KUKA KRL program: EPS_2_25694_RR03_A_20260114065913.src

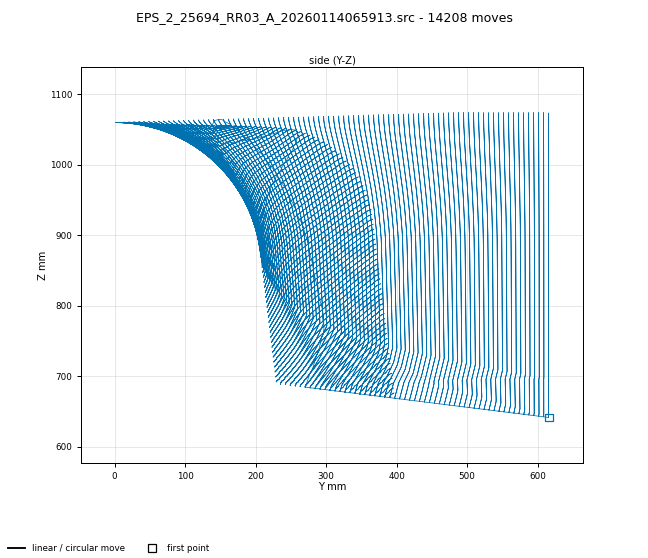
[picture p0: tool path of EPS_2_25694_RR03_A_20260114065913.src, 14208 of 14210 moves have a stored position in this frame; points joined in program order, loops and branches not executed]
&ACCESS RVP
&REL 4
&COMMENT QRS 19112012
&PARAM EDITMASK = *
DEF PART()
EXT BAS (BAS_COMMAND :IN,REAL :IN )
INT I
BAS (#INITMOV,0 )

;KUKA QRS Post kuka4.cps  Date:22-06-2017 !

File_ID=2964

QRS_PRE_INIT()

;Init var - Until changes are made in qrs_pre_init
Outlet_Square_prg=0
Inlet_1_Square_prg=0
Inlet_2_Square_prg=0
Inlet_3_Square_prg=0
Inlet_4_Square_prg=0
Inlet_5_Square_prg=0

Outlet_1={X 0.000, Y 484.060, Z 891.000, B 0.000, E1 0.000 }
Inlet_1={X 0.000, Y 496.780, Z 866.000, B 0.000, E1 180.000 }
Outlet_1_type=366
Inlet_1_type=0
;QRS#1=Sidecore dimensions
;QRS#2=375-15" PVC SDR 35
;QRS#3=DeadEnd 366
;QRS#4=
;QRS#5=
;QRS#6=
;QRS#7=
;QRS#8=
;QRS#9=20Y PSX
;QRS#10=

;QRS#11=
;QRS#12=
;QRS#13=
;QRS#14=
;QRS#15=
;QRS#16=1220x127x1372 4,5'
;QRS#17=EPS Height
;QRS#18=1074
;QRS#19=*
;QRS#20= UPDATED VERSION 22-06-2017
;QRS#21=*
Outlet_Square=0250
Inlet_1_Square=00
Inlet_2_Square=0
Inlet_3_Square=0
Inlet_4_Square=0
Inlet_5_Square=0
Mill_Square=1
Outlet_Square_Prg=252
Inlet_1_Square_prg=0

QRS_INIT()

$ADVANCE=5

; T1
PTP {E1 173.414,E2 173.414}
PTP {X 0,Y 615.481,A -85,B 0,C 180,E1 173.414,E2 173.414,E3 0,E4 0,E5 0,E6 0}
QRS_SPEED_INIT()
LIN {X 0,Y 615.481,Z 641.494,A -85,B 0,C 180,E1 173.414,E2 173.414,E3 0,E4 0,E5 0,E6 0} C_VEL
LIN {X 0,Y 615.482,Z 641.499,A -85,B 0,C 180,E1 170.801,E2 170.801} C_VEL
LIN {X 0,Y 615.492,Z 641.513,A -85,B 0,C 180,E1 168.14,E2 168.14} C_VEL
LIN {X 0,Y 615.474,Z 641.499,A -85,B 0,C 180,E1 165.451,E2 165.451} C_VEL
LIN {X 0,Y 615.49,Z 641.493,A -85,B 0,C 180,E1 162.73,E2 162.73} C_VEL
LIN {X 0,Y 615.49,Z 641.509,A -85,B 0,C 180,E1 159.968,E2 159.968} C_VEL
LIN {X 0,Y 615.475,Z 641.5,A -85,B 0,C 180,E1 157.155,E2 157.155} C_VEL
LIN {X 0,Y 615.494,Z 641.492,A -85,B 0,C 180,E1 154.427,E2 154.427} C_VEL
LIN {X 0,Y 615.492,Z 641.512,A -85,B 0,C 180,E1 151.546,E2 151.546} C_VEL
LIN {X 0,Y 615.475,Z 641.502,A -85,B 0,C 180,E1 148.913,E2 148.913} C_VEL
LIN {X 0,Y 615.48,Z 641.495,A -85,B 0,C 180,E1 146.465,E2 146.465} C_VEL
LIN {X 0,Y 615.492,Z 641.491,A -85,B 0,C 180,E1 144.164,E2 144.164} C_VEL
LIN {X 0,Y 615.485,Z 641.494,A -85,B 0,C 180,E1 141.932,E2 141.932} C_VEL
LIN {X 0,Y 615.479,Z 641.503,A -85,B 0,C 180,E1 139.393,E2 139.393} C_VEL
LIN {X 0,Y 615.494,Z 641.508,A -85,B 0,C 180,E1 136.757,E2 136.757} C_VEL
LIN {X 0,Y 615.476,Z 641.496,A -85,B 0,C 180,E1 133.997,E2 133.997} C_VEL
LIN {X 0,Y 615.478,Z 641.502,A -85,B 0,C 180,E1 131.094,E2 131.094} C_VEL
LIN {X 0,Y 615.48,Z 641.505,A -85,B 0,C 180,E1 128.904,E2 128.904} C_VEL
LIN {X 0,Y 615.485,Z 641.514,A -85,B 0,C 180,E1 126.424,E2 126.424} C_VEL
LIN {X 0,Y 615.482,Z 641.494,A -85,B 0,C 180,E1 123.534,E2 123.534} C_VEL
LIN {X 0,Y 615.481,Z 641.496,A -85,B 0,C 180,E1 120.919,E2 120.919} C_VEL
LIN {X 0,Y 615.477,Z 641.506,A -85,B 0,C 180,E1 118.45,E2 118.45} C_VEL
LIN {X 0,Y 615.477,Z 641.505,A -85,B 0,C 180,E1 115.715,E2 115.715} C_VEL
LIN {X 0,Y 615.486,Z 641.493,A -85,B 0,C 180,E1 112.844,E2 112.844} C_VEL
LIN {X 0,Y 615.483,Z 641.507,A -85,B 0,C 180,E1 110.032,E2 110.032} C_VEL
LIN {X 0,Y 615.476,Z 641.503,A -85,B 0,C 180,E1 107.27,E2 107.27} C_VEL
LIN {X 0,Y 615.488,Z 641.492,A -85,B 0,C 180,E1 104.549,E2 104.549} C_VEL
LIN {X 0,Y 615.477,Z 641.504,A -85,B 0,C 180,E1 101.861,E2 101.861} C_VEL
LIN {X 0,Y 615.487,Z 641.508,A -85,B 0,C 180,E1 99.199,E2 99.199} C_VEL
LIN {X 0,Y 615.479,Z 641.496,A -85,B 0,C 180,E1 96.557,E2 96.557} C_VEL
LIN {X 0,Y 615.483,Z 641.495,A -85,B 0,C 180,E1 93.928,E2 93.928} C_VEL
LIN {X 0,Y 615.481,Z 641.507,A -85,B 0,C 180,E1 91.309,E2 91.309} C_VEL
LIN {X 0,Y 615.481,Z 641.507,A -85,B 0,C 180,E1 88.691,E2 88.691} C_VEL
LIN {X 0,Y 615.483,Z 641.495,A -85,B 0,C 180,E1 86.072,E2 86.072} C_VEL
LIN {X 0,Y 615.478,Z 641.497,A -85,B 0,C 180,E1 83.425,E2 83.425} C_VEL
LIN {X 0,Y 615.487,Z 641.508,A -85,B 0,C 180,E1 80.801,E2 80.801} C_VEL
LIN {X 0,Y 615.477,Z 641.504,A -85,B 0,C 180,E1 78.139,E2 78.139} C_VEL
LIN {X 0,Y 615.488,Z 641.492,A -85,B 0,C 180,E1 75.451,E2 75.451} C_VEL
LIN {X 0,Y 615.476,Z 641.503,A -85,B 0,C 180,E1 72.73,E2 72.73} C_VEL
LIN {X 0,Y 615.483,Z 641.507,A -85,B 0,C 180,E1 69.968,E2 69.968} C_VEL
LIN {X 0,Y 615.486,Z 641.493,A -85,B 0,C 180,E1 67.156,E2 67.156} C_VEL
LIN {X 0,Y 615.477,Z 641.505,A -85,B 0,C 180,E1 64.285,E2 64.285} C_VEL
LIN {X 0,Y 615.48,Z 641.505,A -85,B 0,C 180,E1 61.55,E2 61.55} C_VEL
LIN {X 0,Y 615.49,Z 641.492,A -85,B 0,C 180,E1 58.913,E2 58.913} C_VEL
LIN {X 0,Y 615.482,Z 641.494,A -85,B 0,C 180,E1 56.466,E2 56.466} C_VEL
LIN {X 0,Y 615.485,Z 641.514,A -85,B 0,C 180,E1 53.576,E2 53.576} C_VEL
LIN {X 0,Y 615.478,Z 641.501,A -85,B 0,C 180,E1 50.938,E2 50.938} C_VEL
LIN {X 0,Y 615.487,Z 641.494,A -85,B 0,C 180,E1 48.527,E2 48.527} C_VEL
LIN {X 0,Y 615.473,Z 641.499,A -85,B 0,C 180,E1 45.851,E2 45.851} C_VEL
LIN {X 0,Y 615.489,Z 641.513,A -85,B 0,C 180,E1 43.049,E2 43.049} C_VEL
LIN {X 0,Y 615.497,Z 641.49,A -85,B 0,C 180,E1 40.092,E2 40.092} C_VEL
LIN {X 0,Y 615.479,Z 641.503,A -85,B 0,C 180,E1 37.242,E2 37.242} C_VEL
LIN {X 0,Y 615.491,Z 641.512,A -85,B 0,C 180,E1 34.703,E2 34.703} C_VEL
LIN {X 0,Y 615.487,Z 641.493,A -85,B 0,C 180,E1 31.685,E2 31.685} C_VEL
LIN {X 0,Y 615.482,Z 641.494,A -85,B 0,C 180,E1 29.406,E2 29.406} C_VEL
LIN {X 0,Y 615.494,Z 641.513,A -85,B 0,C 180,E1 26.443,E2 26.443} C_VEL
LIN {X 0,Y 615.488,Z 641.494,A -85,B 0,C 180,E1 23.556,E2 23.556} C_VEL
LIN {X 0,Y 615.475,Z 641.5,A -85,B 0,C 180,E1 20.731,E2 20.731} C_VEL
LIN {X 0,Y 615.488,Z 641.51,A -85,B 0,C 180,E1 17.957,E2 17.957} C_VEL
LIN {X 0,Y 615.489,Z 641.493,A -85,B 0,C 180,E1 15.226,E2 15.226} C_VEL
LIN {X 0,Y 615.475,Z 641.498,A -85,B 0,C 180,E1 12.53,E2 12.53} C_VEL
LIN {X 0,Y 615.495,Z 641.509,A -85,B 0,C 180,E1 9.862,E2 9.862} C_VEL
LIN {X 0,Y 615.481,Z 641.501,A -85,B 0,C 180,E1 7.216,E2 7.216} C_VEL
LIN {X 0,Y 615.492,Z 641.492,A -85,B 0,C 180,E1 4.584,E2 4.584} C_VEL
LIN {X 0,Y 615.476,Z 641.5,A -85,B 0,C 180,E1 1.963,E2 1.963} C_VEL
LIN {X 0,Y 615.492,Z 641.514,A -85,B 0,C 180,E1 -0.654,E2 -0.654} C_VEL
LIN {X 0,Y 615.482,Z 641.5,A -85,B 0,C 180,E1 -3.273,E2 -3.273} C_VEL
LIN {X 0,Y 615.486,Z 641.493,A -85,B 0,C 180,E1 -5.899,E2 -5.899} C_VEL
LIN {X 0,Y 615.479,Z 641.501,A -85,B 0,C 180,E1 -8.537,E2 -8.537} C_VEL
LIN {X 0,Y 615.488,Z 641.511,A -85,B 0,C 180,E1 -11.193,E2 -11.193} C_VEL
LIN {X 0,Y 615.493,Z 641.493,A -85,B 0,C 180,E1 -13.941,E2 -13.941} C_VEL
LIN {X 0,Y 615.475,Z 641.497,A -85,B 0,C 180,E1 -16.587,E2 -16.587} C_VEL
LIN {X 0,Y 615.492,Z 641.51,A -85,B 0,C 180,E1 -19.338,E2 -19.338} C_VEL
LIN {X 0,Y 615.491,Z 641.493,A -85,B 0,C 180,E1 -22.35,E2 -22.35} C_VEL
LIN {X 0,Y 615.475,Z 641.498,A -85,B 0,C 180,E1 -24.992,E2 -24.992} C_VEL
LIN {X 0,Y 615.475,Z 641.5,A -85,B 0,C 180,E1 -27.178,E2 -27.178} C_VEL
LIN {X 0,Y 615.495,Z 641.512,A -85,B 0,C 180,E1 -29.798,E2 -29.798} C_VEL
LIN {X 0,Y 615.484,Z 641.499,A -85,B 0,C 180,E1 -32.458,E2 -32.458} C_VEL
LIN {X 0,Y 615.495,Z 641.492,A -85,B 0,C 180,E1 -34.814,E2 -34.814} C_VEL
LIN {X 0,Y 615.479,Z 641.495,A -85,B 0,C 180,E1 -37.243,E2 -37.243} C_VEL
LIN {X 0,Y 615.498,Z 641.506,A -85,B 0,C 180,E1 -40.092,E2 -40.092} C_VEL
LIN {X 0,Y 615.486,Z 641.495,A -85,B 0,C 180,E1 -43.049,E2 -43.049} C_VEL
LIN {X 0,Y 615.473,Z 641.499,A -85,B 0,C 180,E1 -45.851,E2 -45.851} C_VEL
LIN {X 0,Y 615.49,Z 641.511,A -85,B 0,C 180,E1 -48.528,E2 -48.528} C_VEL
LIN {X 0,Y 615.482,Z 641.502,A -85,B 0,C 180,E1 -51.096,E2 -51.096} C_VEL
LIN {X 0,Y 615.485,Z 641.494,A -85,B 0,C 180,E1 -53.576,E2 -53.576} C_VEL
LIN {X 0,Y 615.482,Z 641.5,A -85,B 0,C 180,E1 -56.466,E2 -56.466} C_VEL
LIN {X 0,Y 615.492,Z 641.512,A -85,B 0,C 180,E1 -59.081,E2 -59.081} C_VEL
LIN {X 0,Y 615.499,Z 641.611,A -85,B 0,C 180,E1 -61.157,E2 -61.157} C_VEL
LIN {X 0,Y 615.495,Z 642.282,A -85,B 0,C 180,E1 -61.343,E2 -61.343} C_VEL
LIN {X 0,Y 615.494,Z 664.074,A -85,B 0,C 180,E1 -64.104,E2 -64.104} C_VEL
LIN {X 0,Y 615.485,Z 687.394,A -85,B 0,C 180,E1 -66.978,E2 -66.978} C_VEL
LIN {X 0,Y 615.494,Z 696.002,A -85,B 0,C 180,E1 -67.997,E2 -67.997} C_VEL
LIN {X 0,Y 615.487,Z 889.623,A -85,B 0,C 180,E1 -70.381,E2 -70.381} C_VEL
LIN {X 0,Y 615.478,Z 906.235,A -85,B 0,C 180,E1 -70.641,E2 -70.641} C_VEL
LIN {X 0,Y 615.481,Z 921.941,A -85,B 0,C 180,E1 -71.009,E2 -71.009} C_VEL
LIN {X 0,Y 615.492,Z 937.98,A -85,B 0,C 180,E1 -71.515,E2 -71.515} C_VEL
LIN {X 0,Y 615.487,Z 955.003,A -85,B 0,C 180,E1 -72.215,E2 -72.215} C_VEL
LIN {X 0,Y 615.498,Z 970.011,A -85,B 0,C 180,E1 -72.987,E2 -72.987} C_VEL
LIN {X 0,Y 615.497,Z 983.749,A -85,B 0,C 180,E1 -73.83,E2 -73.83} C_VEL
LIN {X 0,Y 615.496,Z 997.894,A -85,B 0,C 180,E1 -74.859,E2 -74.859} C_VEL
LIN {X 0,Y 615.496,Z 1010.178,A -85,B 0,C 180,E1 -75.911,E2 -75.911} C_VEL
LIN {X 0,Y 615.493,Z 1022.325,A -85,B 0,C 180,E1 -77.135,E2 -77.135} C_VEL
LIN {X 0,Y 615.491,Z 1033.537,A -85,B 0,C 180,E1 -78.474,E2 -78.474} C_VEL
LIN {X 0,Y 615.493,Z 1042.917,A -85,B 0,C 180,E1 -79.806,E2 -79.806} C_VEL
LIN {X 0,Y 615.495,Z 1050.708,A -85,B 0,C 180,E1 -81.133,E2 -81.133} C_VEL
LIN {X 0,Y 615.494,Z 1057.212,A -85,B 0,C 180,E1 -82.455,E2 -82.455} C_VEL
LIN {X 0,Y 615.494,Z 1062.49,A -85,B 0,C 180,E1 -83.773,E2 -83.773} C_VEL
LIN {X 0,Y 615.497,Z 1065.74,A -85,B 0,C 180,E1 -84.759,E2 -84.759} C_VEL
LIN {X 0,Y 615.492,Z 1069.077,A -85,B 0,C 180,E1 -86.072,E2 -86.072} C_VEL
LIN {X 0,Y 615.484,Z 1071.504,A -85,B 0,C 180,E1 -87.382,E2 -87.382} C_VEL
LIN {X 0,Y 615.494,Z 1072.869,A -85,B 0,C 180,E1 -88.691,E2 -88.691} C_VEL
LIN {X 0,Y 615.489,Z 1073.39,A -85,B 0,C 180,E1 -90,E2 -90} C_VEL
LIN {X 0,Y 615.494,Z 1072.869,A -85,B 0,C 180,E1 -91.309,E2 -91.309} C_VEL
LIN {X 0,Y 615.484,Z 1071.504,A -85,B 0,C 180,E1 -92.618,E2 -92.618} C_VEL
LIN {X 0,Y 615.492,Z 1069.077,A -85,B 0,C 180,E1 -93.928,E2 -93.928} C_VEL
LIN {X 0,Y 615.496,Z 1065.74,A -85,B 0,C 180,E1 -95.241,E2 -95.241} C_VEL
LIN {X 0,Y 615.495,Z 1059.981,A -85,B 0,C 180,E1 -96.898,E2 -96.898} C_VEL
LIN {X 0,Y 615.491,Z 1052.502,A -85,B 0,C 180,E1 -98.536,E2 -98.536} C_VEL
LIN {X 0,Y 615.489,Z 1043.967,A -85,B 0,C 180,E1 -100.028,E2 -100.028} C_VEL
LIN {X 0,Y 615.496,Z 1034.768,A -85,B 0,C 180,E1 -101.359,E2 -101.359} C_VEL
LIN {X 0,Y 615.494,Z 1025.294,A -85,B 0,C 180,E1 -102.53,E2 -102.53} C_VEL
LIN {X 0,Y 615.495,Z 1014.218,A -85,B 0,C 180,E1 -103.705,E2 -103.705} C_VEL
LIN {X 0,Y 615.495,Z 1002.119,A -85,B 0,C 180,E1 -104.802,E2 -104.802} C_VEL
LIN {X 0,Y 615.497,Z 987.714,A -85,B 0,C 180,E1 -105.904,E2 -105.904} C_VEL
LIN {X 0,Y 615.497,Z 973.021,A -85,B 0,C 180,E1 -106.842,E2 -106.842} C_VEL
LIN {X 0,Y 615.497,Z 958.52,A -85,B 0,C 180,E1 -107.613,E2 -107.613} C_VEL
LIN {X 0,Y 615.486,Z 943.271,A -85,B 0,C 180,E1 -108.281,E2 -108.281} C_VEL
LIN {X 0,Y 615.488,Z 928.006,A -85,B 0,C 180,E1 -108.818,E2 -108.818} C_VEL
LIN {X 0,Y 615.476,Z 911.542,A -85,B 0,C 180,E1 -109.251,E2 -109.251} C_VEL
LIN {X 0,Y 615.484,Z 895.965,A -85,B 0,C 180,E1 -109.533,E2 -109.533} C_VEL
LIN {X 0,Y 615.492,Z 696.002,A -85,B 0,C 180,E1 -112.003,E2 -112.003} C_VEL
LIN {X 0,Y 615.475,Z 675.734,A -85,B 0,C 180,E1 -114.451,E2 -114.451} C_VEL
LIN {X 0,Y 615.495,Z 653.871,A -85,B 0,C 180,E1 -117.176,E2 -117.176} C_VEL
LIN {X 0,Y 615.496,Z 641.859,A -85,B 0,C 180,E1 -118.727,E2 -118.727} C_VEL
LIN {X 0,Y 615.478,Z 641.5,A -85,B 0,C 180,E1 -119.406,E2 -119.406} C_VEL
LIN {X 0,Y 615.473,Z 641.498,A -85,B 0,C 180,E1 -121.685,E2 -121.685} C_VEL
LIN {X 0,Y 615.479,Z 641.495,A -85,B 0,C 180,E1 -124.021,E2 -124.021} C_VEL
LIN {X 0,Y 615.486,Z 641.505,A -85,B 0,C 180,E1 -126.937,E2 -126.937} C_VEL
LIN {X 0,Y 615.484,Z 641.501,A -85,B 0,C 180,E1 -129.749,E2 -129.749} C_VEL
LIN {X 0,Y 615.479,Z 641.494,A -85,B 0,C 180,E1 -132.352,E2 -132.352} C_VEL
LIN {X 0,Y 615.485,Z 641.5,A -85,B 0,C 180,E1 -135.067,E2 -135.067} C_VEL
LIN {X 0,Y 615.495,Z 641.503,A -85,B 0,C 180,E1 -137.917,E2 -137.917} C_VEL
LIN {X 0,Y 615.479,Z 641.5,A -85,B 0,C 180,E1 -140.249,E2 -140.249} C_VEL
LIN {X 0,Y 615.487,Z 641.493,A -85,B 0,C 180,E1 -143.061,E2 -143.061} C_VEL
LIN {X 0,Y 615.494,Z 641.514,A -85,B 0,C 180,E1 -145.979,E2 -145.979} C_VEL
LIN {X 0,Y 615.488,Z 641.506,A -85,B 0,C 180,E1 -148.315,E2 -148.315} C_VEL
LIN {X 0,Y 615.482,Z 641.501,A -85,B 0,C 180,E1 -150.593,E2 -150.593} C_VEL
LIN {X 0,Y 615.474,Z 641.498,A -85,B 0,C 180,E1 -152.954,E2 -152.954} C_VEL
LIN {X 0,Y 615.489,Z 641.495,A -85,B 0,C 180,E1 -155.728,E2 -155.728} C_VEL
LIN {X 0,Y 615.492,Z 641.511,A -85,B 0,C 180,E1 -158.568,E2 -158.568} C_VEL
LIN {X 0,Y 615.476,Z 641.496,A -85,B 0,C 180,E1 -161.394,E2 -161.394} C_VEL
LIN {X 0,Y 615.487,Z 641.496,A -85,B 0,C 180,E1 -164.095,E2 -164.095} C_VEL
LIN {X 0,Y 615.495,Z 641.513,A -85,B 0,C 180,E1 -166.799,E2 -166.799} C_VEL
LIN {X 0,Y 615.474,Z 641.5,A -85,B 0,C 180,E1 -169.473,E2 -169.473} C_VEL
LIN {X 0,Y 615.486,Z 641.493,A -85,B 0,C 180,E1 -172.124,E2 -172.124} C_VEL
LIN {X 0,Y 615.482,Z 641.502,A -85,B 0,C 180,E1 -174.759,E2 -174.759} C_VEL
LIN {X 0,Y 615.495,Z 641.508,A -85,B 0,C 180,E1 -177.382,E2 -177.382} C_VEL
LIN {X 0,Y 615.475,Z 641.498,A -85,B 0,C 180,E1 -180,E2 -180} C_VEL
LIN {X 0,Y 615.492,Z 641.492,A -85,B 0,C 180,E1 -182.618,E2 -182.618} C_VEL
LIN {X 0,Y 615.482,Z 641.504,A -85,B 0,C 180,E1 -185.241,E2 -185.241} C_VEL
LIN {X 0,Y 615.481,Z 641.494,A -85,B 0,C 180,E1 -186.586,E2 -186.586} C_VEL
LIN {X 0,Y 614.804,Z 641.649,A -85,B 0,C 180,E1 -187.132,E2 -187.132} C_VEL
LIN {X 0,Y 611.968,Z 642.066,A -85,B 0,C 180,E1 -188.018,E2 -188.018} C_VEL
LIN {X 0,Y 609.577,Z 642.375,A -85,B 0,C 180,E1 -188.731,E2 -188.731} C_VEL
LIN {X 0,Y 608.545,Z 642.492,A -85,B 0,C 180,E1 -189.28,E2 -189.28} C_VEL
LIN {X 0,Y 608.458,Z 642.502,A -85,B 0,C 180,E1 -189.466,E2 -189.466} C_VEL
LIN {X 0,Y 608.462,Z 642.506,A -85,B 0,C 180,E1 -192,E2 -192} C_VEL
LIN {X 0,Y 608.466,Z 642.497,A -85,B 0,C 180,E1 -194.72,E2 -194.72} C_VEL
LIN {X 0,Y 608.455,Z 642.5,A -85,B 0,C 180,E1 -197.476,E2 -197.476} C_VEL
LIN {X 0,Y 608.461,Z 642.508,A -85,B 0,C 180,E1 -200.274,E2 -200.274} C_VEL
LIN {X 0,Y 608.482,Z 642.502,A -85,B 0,C 180,E1 -202.485,E2 -202.485} C_VEL
LIN {X 0,Y 608.449,Z 642.499,A -85,B 0,C 180,E1 -205.301,E2 -205.301} C_VEL
LIN {X 0,Y 608.441,Z 642.499,A -85,B 0,C 180,E1 -207.518,E2 -207.518} C_VEL
LIN {X 0,Y 608.465,Z 642.498,A -85,B 0,C 180,E1 -209.974,E2 -209.974} C_VEL
LIN {X 0,Y 608.458,Z 642.507,A -85,B 0,C 180,E1 -212.524,E2 -212.524} C_VEL
LIN {X 0,Y 608.443,Z 642.502,A -85,B 0,C 180,E1 -215.277,E2 -215.277} C_VEL
LIN {X 0,Y 608.465,Z 642.497,A -85,B 0,C 180,E1 -217.746,E2 -217.746} C_VEL
LIN {X 0,Y 608.471,Z 642.498,A -85,B 0,C 180,E1 -220.333,E2 -220.333} C_VEL
LIN {X 0,Y 608.48,Z 642.503,A -85,B 0,C 180,E1 -223.311,E2 -223.311} C_VEL
LIN {X 0,Y 608.461,Z 642.498,A -85,B 0,C 180,E1 -226.131,E2 -226.131} C_VEL
LIN {X 0,Y 608.45,Z 642.502,A -85,B 0,C 180,E1 -228.824,E2 -228.824} C_VEL
LIN {X 0,Y 608.461,Z 642.509,A -85,B 0,C 180,E1 -231.413,E2 -231.413} C_VEL
LIN {X 0,Y 608.469,Z 642.501,A -85,B 0,C 180,E1 -233.951,E2 -233.951} C_VEL
LIN {X 0,Y 608.459,Z 642.499,A -85,B 0,C 180,E1 -236.33,E2 -236.33} C_VEL
LIN {X 0,Y 608.473,Z 642.496,A -85,B 0,C 180,E1 -238.727,E2 -238.727} C_VEL
LIN {X 0,Y 608.464,Z 642.501,A -85,B 0,C 180,E1 -241.381,E2 -241.381} C_VEL
LIN {X 0,Y 608.437,Z 642.513,A -85,B 0,C 180,E1 -243.965,E2 -243.965} C_VEL
LIN {X 0,Y 608.466,Z 642.507,A -85,B 0,C 180,E1 -246.156,E2 -246.156} C_VEL
LIN {X 0,Y 608.455,Z 642.498,A -85,B 0,C 180,E1 -249.019,E2 -249.019} C_VEL
LIN {X 0,Y 608.447,Z 642.503,A -85,B 0,C 180,E1 -251.829,E2 -251.829} C_VEL
LIN {X 0,Y 608.463,Z 642.505,A -85,B 0,C 180,E1 -254.594,E2 -254.594} C_VEL
LIN {X 0,Y 608.473,Z 642.496,A -85,B 0,C 180,E1 -257.323,E2 -257.323} C_VEL
LIN {X 0,Y 608.449,Z 642.501,A -85,B 0,C 180,E1 -260.023,E2 -260.023} C_VEL
LIN {X 0,Y 608.461,Z 642.51,A -85,B 0,C 180,E1 -262.701,E2 -262.701} C_VEL
LIN {X 0,Y 608.446,Z 642.502,A -85,B 0,C 180,E1 -265.362,E2 -265.362} C_VEL
LIN {X 0,Y 608.46,Z 642.498,A -85,B 0,C 180,E1 -268.014,E2 -268.014} C_VEL
LIN {X 0,Y 608.47,Z 642.502,A -85,B 0,C 180,E1 -270.662,E2 -270.662} C_VEL
LIN {X 0,Y 608.48,Z 642.504,A -85,B 0,C 180,E1 -273.311,E2 -273.311} C_VEL
LIN {X 0,Y 608.452,Z 642.5,A -85,B 0,C 180,E1 -275.967,E2 -275.967} C_VEL
LIN {X 0,Y 608.454,Z 642.5,A -85,B 0,C 180,E1 -278.636,E2 -278.636} C_VEL
LIN {X 0,Y 608.472,Z 642.506,A -85,B 0,C 180,E1 -281.324,E2 -281.324} C_VEL
LIN {X 0,Y 608.464,Z 642.501,A -85,B 0,C 180,E1 -284.037,E2 -284.037} C_VEL
LIN {X 0,Y 608.475,Z 642.496,A -85,B 0,C 180,E1 -286.783,E2 -286.783} C_VEL
LIN {X 0,Y 608.443,Z 642.507,A -85,B 0,C 180,E1 -289.57,E2 -289.57} C_VEL
LIN {X 0,Y 608.47,Z 642.5,A -85,B 0,C 180,E1 -292.405,E2 -292.405} C_VEL
LIN {X 0,Y 608.452,Z 642.501,A -85,B 0,C 180,E1 -294.57,E2 -294.57} C_VEL
LIN {X 0,Y 608.482,Z 642.495,A -85,B 0,C 180,E1 -297.209,E2 -297.209} C_VEL
LIN {X 0,Y 608.464,Z 642.504,A -85,B 0,C 180,E1 -299.972,E2 -299.972} C_VEL
LIN {X 0,Y 608.46,Z 642.506,A -85,B 0,C 180,E1 -302.523,E2 -302.523} C_VEL
LIN {X 0,Y 608.438,Z 642.501,A -85,B 0,C 180,E1 -305.277,E2 -305.277} C_VEL
LIN {X 0,Y 608.46,Z 642.498,A -85,B 0,C 180,E1 -307.746,E2 -307.746} C_VEL
LIN {X 0,Y 608.447,Z 642.505,A -85,B 0,C 180,E1 -310.329,E2 -310.329} C_VEL
LIN {X 0,Y 608.466,Z 642.499,A -85,B 0,C 180,E1 -313.309,E2 -313.309} C_VEL
LIN {X 0,Y 608.468,Z 642.497,A -85,B 0,C 180,E1 -316.131,E2 -316.131} C_VEL
LIN {X 0,Y 608.456,Z 642.507,A -85,B 0,C 180,E1 -318.824,E2 -318.824} C_VEL
LIN {X 0,Y 608.471,Z 642.502,A -85,B 0,C 180,E1 -321.413,E2 -321.413} C_VEL
LIN {X 0,Y 608.471,Z 642.496,A -85,B 0,C 180,E1 -323.949,E2 -323.949} C_VEL
LIN {X 0,Y 608.458,Z 642.498,A -85,B 0,C 180,E1 -326.329,E2 -326.329} C_VEL
LIN {X 0,Y 608.466,Z 642.498,A -85,B 0,C 180,E1 -328.727,E2 -328.727} C_VEL
LIN {X 0,Y 608.474,Z 642.505,A -85,B 0,C 180,E1 -331.377,E2 -331.377} C_VEL
LIN {X 0,Y 608.471,Z 642.498,A -85,B 0,C 180,E1 -334.276,E2 -334.276} C_VEL
LIN {X 0,Y 608.444,Z 642.5,A -85,B 0,C 180,E1 -336.876,E2 -336.876} C_VEL
LIN {X 0,Y 608.459,Z 642.501,A -85,B 0,C 180,E1 -339.32,E2 -339.32} C_VEL
LIN {X 0,Y 608.448,Z 642.51,A -85,B 0,C 180,E1 -341.828,E2 -341.828} C_VEL
LIN {X 0,Y 608.472,Z 642.498,A -85,B 0,C 180,E1 -344.594,E2 -344.594} C_VEL
LIN {X 0,Y 608.466,Z 642.497,A -85,B 0,C 180,E1 -347.323,E2 -347.323} C_VEL
LIN {X 0,Y 608.46,Z 642.505,A -85,B 0,C 180,E1 -350.023,E2 -350.023} C_VEL
LIN {X 0,Y 608.475,Z 642.501,A -85,B 0,C 180,E1 -352.701,E2 -352.701} C_VEL
LIN {X 0,Y 608.46,Z 642.498,A -85,B 0,C 180,E1 -355.363,E2 -355.363} C_VEL
LIN {X 0,Y 608.447,Z 642.501,A -85,B 0,C 180,E1 -358.014,E2 -358.014} C_VEL
LIN {X 0,Y 608.484,Z 642.507,A -85,B 0,C 180,E1 -360.662,E2 -360.662} C_VEL
LIN {X 0,Y 608.474,Z 642.498,A -85,B 0,C 180,E1 -363.311,E2 -363.311} C_VEL
LIN {X 0,Y 608.481,Z 642.495,A -85,B 0,C 180,E1 -365.967,E2 -365.967} C_VEL
LIN {X 0,Y 608.45,Z 642.504,A -85,B 0,C 180,E1 -368.636,E2 -368.636} C_VEL
LIN {X 0,Y 608.474,Z 642.503,A -85,B 0,C 180,E1 -371.324,E2 -371.324} C_VEL
LIN {X 0,Y 608.458,Z 642.498,A -85,B 0,C 180,E1 -374.038,E2 -374.038} C_VEL
LIN {X 0,Y 608.467,Z 642.499,A -85,B 0,C 180,E1 -376.784,E2 -376.784} C_VEL
LIN {X 0,Y 608.454,Z 642.508,A -85,B 0,C 180,E1 -379.571,E2 -379.571} C_VEL
LIN {X 0,Y 608.468,Z 642.496,A -85,B 0,C 180,E1 -382.482,E2 -382.482} C_VEL
LIN {X 0,Y 608.448,Z 642.504,A -85,B 0,C 180,E1 -385.301,E2 -385.301} C_VEL
LIN {X 0,Y 608.444,Z 642.507,A -85,B 0,C 180,E1 -387.518,E2 -387.518} C_VEL
LIN {X 0,Y 608.471,Z 642.506,A -85,B 0,C 180,E1 -389.975,E2 -389.975} C_VEL
LIN {X 0,Y 608.457,Z 642.5,A -85,B 0,C 180,E1 -392.524,E2 -392.524} C_VEL
LIN {X 0,Y 608.443,Z 642.5,A -85,B 0,C 180,E1 -395.278,E2 -395.278} C_VEL
LIN {X 0,Y 608.469,Z 642.5,A -85,B 0,C 180,E1 -397.746,E2 -397.746} C_VEL
LIN {X 0,Y 608.474,Z 642.507,A -85,B 0,C 180,E1 -400.333,E2 -400.333} C_VEL
LIN {X 0,Y 608.48,Z 642.495,A -85,B 0,C 180,E1 -403.311,E2 -403.311} C_VEL
LIN {X 0,Y 608.462,Z 642.502,A -85,B 0,C 180,E1 -406.131,E2 -406.131} C_VEL
LIN {X 0,Y 608.454,Z 642.506,A -85,B 0,C 180,E1 -408.825,E2 -408.825} C_VEL
LIN {X 0,Y 608.463,Z 642.498,A -85,B 0,C 180,E1 -411.413,E2 -411.413} C_VEL
LIN {X 0,Y 608.471,Z 642.496,A -85,B 0,C 180,E1 -413.951,E2 -413.951} C_VEL
LIN {X 0,Y 608.459,Z 642.5,A -85,B 0,C 180,E1 -416.33,E2 -416.33} C_VEL
LIN {X 0,Y 608.476,Z 642.501,A -85,B 0,C 180,E1 -418.728,E2 -418.728} C_VEL
LIN {X 0,Y 608.508,Z 642.684,A -85,B 0,C 180,E1 -421.015,E2 -421.015} C_VEL
LIN {X 0,Y 608.742,Z 646.926,A -85,B 0,C 180,E1 -421.605,E2 -421.605} C_VEL
LIN {X 0,Y 608.689,Z 667.591,A -85,B 0,C 180,E1 -424.236,E2 -424.236} C_VEL
LIN {X 0,Y 608.628,Z 690.455,A -85,B 0,C 180,E1 -427.082,E2 -427.082} C_VEL
LIN {X 0,Y 608.66,Z 695.999,A -85,B 0,C 180,E1 -427.737,E2 -427.737} C_VEL
LIN {X 0,Y 608.923,Z 700.026,A -85,B 0,C 180,E1 -427.814,E2 -427.814} C_VEL
LIN {X 0,Y 608.793,Z 898.977,A -85,B 0,C 180,E1 -430.288,E2 -430.288} C_VEL
LIN {X 0,Y 608.766,Z 915.2,A -85,B 0,C 180,E1 -430.616,E2 -430.616} C_VEL
LIN {X 0,Y 608.751,Z 931.96,A -85,B 0,C 180,E1 -431.097,E2 -431.097} C_VEL
LIN {X 0,Y 608.685,Z 947.354,A -85,B 0,C 180,E1 -431.672,E2 -431.672} C_VEL
LIN {X 0,Y 608.673,Z 962.02,A -85,B 0,C 180,E1 -432.357,E2 -432.357} C_VEL
LIN {X 0,Y 608.616,Z 975.841,A -85,B 0,C 180,E1 -433.135,E2 -433.135} C_VEL
LIN {X 0,Y 608.578,Z 990.054,A -85,B 0,C 180,E1 -434.082,E2 -434.082} C_VEL
LIN {X 0,Y 608.556,Z 1003.132,A -85,B 0,C 180,E1 -435.111,E2 -435.111} C_VEL
LIN {X 0,Y 608.515,Z 1016.01,A -85,B 0,C 180,E1 -436.305,E2 -436.305} C_VEL
LIN {X 0,Y 608.491,Z 1026.914,A -85,B 0,C 180,E1 -437.493,E2 -437.493} C_VEL
LIN {X 0,Y 608.488,Z 1036.208,A -85,B 0,C 180,E1 -438.677,E2 -438.677} C_VEL
LIN {X 0,Y 608.464,Z 1045.26,A -85,B 0,C 180,E1 -440.023,E2 -440.023} C_VEL
LIN {X 0,Y 608.445,Z 1052.859,A -85,B 0,C 180,E1 -441.364,E2 -441.364} C_VEL
LIN {X 0,Y 608.44,Z 1060.467,A -85,B 0,C 180,E1 -443.034,E2 -443.034} C_VEL
LIN {X 0,Y 608.439,Z 1066.245,A -85,B 0,C 180,E1 -444.698,E2 -444.698} C_VEL
LIN {X 0,Y 608.429,Z 1069.633,A -85,B 0,C 180,E1 -446.026,E2 -446.026} C_VEL
LIN {X 0,Y 608.412,Z 1072.086,A -85,B 0,C 180,E1 -447.352,E2 -447.352} C_VEL
LIN {X 0,Y 608.446,Z 1073.477,A -85,B 0,C 180,E1 -448.676,E2 -448.676} C_VEL
LIN {X 0,Y 608.429,Z 1074,A -85,B 0,C 180,E1 -450,E2 -450} C_VEL
LIN {X 0,Y 608.446,Z 1073.477,A -85,B 0,C 180,E1 -451.324,E2 -451.324} C_VEL
LIN {X 0,Y 608.412,Z 1072.086,A -85,B 0,C 180,E1 -452.648,E2 -452.648} C_VEL
LIN {X 0,Y 608.429,Z 1069.633,A -85,B 0,C 180,E1 -453.974,E2 -453.974} C_VEL
LIN {X 0,Y 608.438,Z 1066.245,A -85,B 0,C 180,E1 -455.302,E2 -455.302} C_VEL
LIN {X 0,Y 608.44,Z 1060.467,A -85,B 0,C 180,E1 -456.966,E2 -456.966} C_VEL
LIN {X 0,Y 608.445,Z 1052.859,A -85,B 0,C 180,E1 -458.636,E2 -458.636} C_VEL
LIN {X 0,Y 608.458,Z 1044.248,A -85,B 0,C 180,E1 -460.145,E2 -460.145} C_VEL
LIN {X 0,Y 608.465,Z 1034.969,A -85,B 0,C 180,E1 -461.492,E2 -461.492} C_VEL
LIN {X 0,Y 608.49,Z 1025.424,A -85,B 0,C 180,E1 -462.676,E2 -462.676} C_VEL
LIN {X 0,Y 608.519,Z 1013.976,A -85,B 0,C 180,E1 -463.896,E2 -463.896} C_VEL
LIN {X 0,Y 608.553,Z 1002.147,A -85,B 0,C 180,E1 -464.975,E2 -464.975} C_VEL
LIN {X 0,Y 608.598,Z 988.893,A -85,B 0,C 180,E1 -466.004,E2 -466.004} C_VEL
LIN {X 0,Y 608.616,Z 975.841,A -85,B 0,C 180,E1 -466.865,E2 -466.865} C_VEL
LIN {X 0,Y 608.673,Z 962.02,A -85,B 0,C 180,E1 -467.643,E2 -467.643} C_VEL
LIN {X 0,Y 608.685,Z 947.354,A -85,B 0,C 180,E1 -468.328,E2 -468.328} C_VEL
LIN {X 0,Y 608.751,Z 931.96,A -85,B 0,C 180,E1 -468.903,E2 -468.903} C_VEL
LIN {X 0,Y 608.766,Z 915.2,A -85,B 0,C 180,E1 -469.384,E2 -469.384} C_VEL
LIN {X 0,Y 608.793,Z 898.977,A -85,B 0,C 180,E1 -469.712,E2 -469.712} C_VEL
LIN {X 0,Y 608.881,Z 697.149,A -85,B 0,C 180,E1 -472.224,E2 -472.224} C_VEL
LIN {X 0,Y 608.632,Z 695.447,A -85,B 0,C 180,E1 -472.309,E2 -472.309} C_VEL
LIN {X 0,Y 608.682,Z 672.819,A -85,B 0,C 180,E1 -475.107,E2 -475.107} C_VEL
LIN {X 0,Y 608.74,Z 649.498,A -85,B 0,C 180,E1 -478.064,E2 -478.064} C_VEL
LIN {X 0,Y 608.582,Z 643.159,A -85,B 0,C 180,E1 -478.896,E2 -478.896} C_VEL
LIN {X 0,Y 608.489,Z 642.596,A -85,B 0,C 180,E1 -479.018,E2 -479.018} C_VEL
LIN {X 0,Y 608.474,Z 642.501,A -85,B 0,C 180,E1 -481.315,E2 -481.315} C_VEL
LIN {X 0,Y 608.468,Z 642.498,A -85,B 0,C 180,E1 -483.734,E2 -483.734} C_VEL
LIN {X 0,Y 608.471,Z 642.496,A -85,B 0,C 180,E1 -486.089,E2 -486.089} C_VEL
LIN {X 0,Y 608.463,Z 642.498,A -85,B 0,C 180,E1 -488.587,E2 -488.587} C_VEL
LIN {X 0,Y 608.463,Z 642.509,A -85,B 0,C 180,E1 -491.342,E2 -491.342} C_VEL
LIN {X 0,Y 608.444,Z 642.5,A -85,B 0,C 180,E1 -494.263,E2 -494.263} C_VEL
LIN {X 0,Y 608.456,Z 642.5,A -85,B 0,C 180,E1 -497.041,E2 -497.041} C_VEL
LIN {X 0,Y 608.459,Z 642.509,A -85,B 0,C 180,E1 -499.697,E2 -499.697} C_VEL
LIN {X 0,Y 608.469,Z 642.5,A -85,B 0,C 180,E1 -502.254,E2 -502.254} C_VEL
LIN {X 0,Y 608.483,Z 642.495,A -85,B 0,C 180,E1 -505.088,E2 -505.088} C_VEL
LIN {X 0,Y 608.464,Z 642.506,A -85,B 0,C 180,E1 -507.905,E2 -507.905} C_VEL
LIN {X 0,Y 608.478,Z 642.505,A -85,B 0,C 180,E1 -510.221,E2 -510.221} C_VEL
LIN {X 0,Y 608.468,Z 642.499,A -85,B 0,C 180,E1 -512.792,E2 -512.792} C_VEL
LIN {X 0,Y 608.449,Z 642.499,A -85,B 0,C 180,E1 -515.429,E2 -515.429} C_VEL
LIN {X 0,Y 608.47,Z 642.505,A -85,B 0,C 180,E1 -518.308,E2 -518.308} C_VEL
LIN {X 0,Y 608.46,Z 642.499,A -85,B 0,C 180,E1 -521.283,E2 -521.283} C_VEL
LIN {X 0,Y 608.478,Z 642.496,A -85,B 0,C 180,E1 -523.907,E2 -523.907} C_VEL
LIN {X 0,Y 608.47,Z 642.505,A -85,B 0,C 180,E1 -526.644,E2 -526.644} C_VEL
LIN {X 0,Y 608.458,Z 642.502,A -85,B 0,C 180,E1 -529.35,E2 -529.35} C_VEL
LIN {X 0,Y 608.475,Z 642.495,A -85,B 0,C 180,E1 -532.033,E2 -532.033} C_VEL
LIN {X 0,Y 608.461,Z 642.501,A -85,B 0,C 180,E1 -534.698,E2 -534.698} C_VEL
LIN {X 0,Y 608.483,Z 642.505,A -85,B 0,C 180,E1 -537.352,E2 -537.352} C_VEL
LIN {X 0,Y 608.465,Z 642.498,A -85,B 0,C 180,E1 -540,E2 -540} C_VEL
LIN {X 0,Y 608.481,Z 642.495,A -85,B 0,C 180,E1 -542.648,E2 -542.648} C_VEL
LIN {X 0,Y 608.461,Z 642.504,A -85,B 0,C 180,E1 -545.302,E2 -545.302} C_VEL
LIN {X 0,Y 608.475,Z 642.502,A -85,B 0,C 180,E1 -547.967,E2 -547.967} C_VEL
LIN {X 0,Y 608.458,Z 642.502,A -85,B 0,C 180,E1 -549.466,E2 -549.466} C_VEL
LIN {X 0,Y 607.783,Z 642.59,A -85,B 0,C 180,E1 -550.019,E2 -550.019} C_VEL
LIN {X 0,Y 604.929,Z 642.946,A -85,B 0,C 180,E1 -550.916,E2 -550.916} C_VEL
LIN {X 0,Y 602.523,Z 643.245,A -85,B 0,C 180,E1 -551.637,E2 -551.637} C_VEL
LIN {X 0,Y 601.489,Z 643.371,A -85,B 0,C 180,E1 -552.194,E2 -552.194} C_VEL
LIN {X 0,Y 601.405,Z 643.378,A -85,B 0,C 180,E1 -552.383,E2 -552.383} C_VEL
LIN {X 0,Y 601.423,Z 643.374,A -85,B 0,C 180,E1 -554.897,E2 -554.897} C_VEL
LIN {X 0,Y 601.425,Z 643.374,A -85,B 0,C 180,E1 -556.986,E2 -556.986} C_VEL
LIN {X 0,Y 601.406,Z 643.381,A -85,B 0,C 180,E1 -559.809,E2 -559.809} C_VEL
LIN {X 0,Y 601.444,Z 643.376,A -85,B 0,C 180,E1 -562.681,E2 -562.681} C_VEL
LIN {X 0,Y 601.398,Z 643.38,A -85,B 0,C 180,E1 -564.878,E2 -564.878} C_VEL
LIN {X 0,Y 601.416,Z 643.376,A -85,B 0,C 180,E1 -567.867,E2 -567.867} C_VEL
LIN {X 0,Y 601.437,Z 643.375,A -85,B 0,C 180,E1 -570.163,E2 -570.163} C_VEL
LIN {X 0,Y 601.417,Z 643.386,A -85,B 0,C 180,E1 -572.717,E2 -572.717} C_VEL
LIN {X 0,Y 601.412,Z 643.379,A -85,B 0,C 180,E1 -575.116,E2 -575.116} C_VEL
LIN {X 0,Y 601.427,Z 643.376,A -85,B 0,C 180,E1 -577.419,E2 -577.419} C_VEL
LIN {X 0,Y 601.41,Z 643.376,A -85,B 0,C 180,E1 -579.995,E2 -579.995} C_VEL
LIN {X 0,Y 601.429,Z 643.378,A -85,B 0,C 180,E1 -582.668,E2 -582.668} C_VEL
LIN {X 0,Y 601.416,Z 643.382,A -85,B 0,C 180,E1 -585.483,E2 -585.483} C_VEL
LIN {X 0,Y 601.418,Z 643.375,A -85,B 0,C 180,E1 -588.407,E2 -588.407} C_VEL
LIN {X 0,Y 601.427,Z 643.376,A -85,B 0,C 180,E1 -590.876,E2 -590.876} C_VEL
LIN {X 0,Y 601.436,Z 643.381,A -85,B 0,C 180,E1 -593.734,E2 -593.734} C_VEL
LIN {X 0,Y 601.423,Z 643.374,A -85,B 0,C 180,E1 -596.687,E2 -596.687} C_VEL
LIN {X 0,Y 601.428,Z 643.375,A -85,B 0,C 180,E1 -599.059,E2 -599.059} C_VEL
LIN {X 0,Y 601.424,Z 643.378,A -85,B 0,C 180,E1 -601.374,E2 -601.374} C_VEL
LIN {X 0,Y 601.399,Z 643.384,A -85,B 0,C 180,E1 -603.637,E2 -603.637} C_VEL
LIN {X 0,Y 601.417,Z 643.378,A -85,B 0,C 180,E1 -606.59,E2 -606.59} C_VEL
LIN {X 0,Y 601.429,Z 643.375,A -85,B 0,C 180,E1 -609.479,E2 -609.479} C_VEL
LIN {X 0,Y 601.392,Z 643.39,A -85,B 0,C 180,E1 -612.312,E2 -612.312} C_VEL
LIN {X 0,Y 601.409,Z 643.388,A -85,B 0,C 180,E1 -614.409,E2 -614.409} C_VEL
LIN {X 0,Y 601.416,Z 643.376,A -85,B 0,C 180,E1 -617.172,E2 -617.172} C_VEL
LIN {X 0,Y 601.427,Z 643.375,A -85,B 0,C 180,E1 -619.905,E2 -619.905} C_VEL
LIN {X 0,Y 601.437,Z 643.383,A -85,B 0,C 180,E1 -622.615,E2 -622.615} C_VEL
LIN {X 0,Y 601.416,Z 643.379,A -85,B 0,C 180,E1 -625.308,E2 -625.308} C_VEL
LIN {X 0,Y 601.429,Z 643.374,A -85,B 0,C 180,E1 -627.991,E2 -627.991} C_VEL
LIN {X 0,Y 601.442,Z 643.377,A -85,B 0,C 180,E1 -630.67,E2 -630.67} C_VEL
LIN {X 0,Y 601.432,Z 643.381,A -85,B 0,C 180,E1 -633.349,E2 -633.349} C_VEL
LIN {X 0,Y 601.406,Z 643.377,A -85,B 0,C 180,E1 -636.037,E2 -636.037} C_VEL
LIN {X 0,Y 601.434,Z 643.375,A -85,B 0,C 180,E1 -638.737,E2 -638.737} C_VEL
LIN {X 0,Y 601.43,Z 643.385,A -85,B 0,C 180,E1 -641.458,E2 -641.458} C_VEL
LIN {X 0,Y 601.415,Z 643.377,A -85,B 0,C 180,E1 -644.205,E2 -644.205} C_VEL
LIN {X 0,Y 601.429,Z 643.375,A -85,B 0,C 180,E1 -646.985,E2 -646.985} C_VEL
LIN {X 0,Y 601.4,Z 643.389,A -85,B 0,C 180,E1 -649.809,E2 -649.809} C_VEL
LIN {X 0,Y 601.409,Z 643.377,A -85,B 0,C 180,E1 -652.605,E2 -652.605} C_VEL
LIN {X 0,Y 601.399,Z 643.378,A -85,B 0,C 180,E1 -654.878,E2 -654.878} C_VEL
LIN {X 0,Y 601.419,Z 643.382,A -85,B 0,C 180,E1 -657.867,E2 -657.867} C_VEL
LIN {X 0,Y 601.442,Z 643.383,A -85,B 0,C 180,E1 -660.162,E2 -660.162} C_VEL
LIN {X 0,Y 601.421,Z 643.379,A -85,B 0,C 180,E1 -662.716,E2 -662.716} C_VEL
LIN {X 0,Y 601.404,Z 643.378,A -85,B 0,C 180,E1 -665.114,E2 -665.114} C_VEL
LIN {X 0,Y 601.427,Z 643.374,A -85,B 0,C 180,E1 -667.418,E2 -667.418} C_VEL
LIN {X 0,Y 601.404,Z 643.378,A -85,B 0,C 180,E1 -669.994,E2 -669.994} C_VEL
LIN {X 0,Y 601.404,Z 643.388,A -85,B 0,C 180,E1 -672.67,E2 -672.67} C_VEL
LIN {X 0,Y 601.416,Z 643.377,A -85,B 0,C 180,E1 -675.482,E2 -675.482} C_VEL
LIN {X 0,Y 601.422,Z 643.377,A -85,B 0,C 180,E1 -678.405,E2 -678.405} C_VEL
LIN {X 0,Y 601.433,Z 643.381,A -85,B 0,C 180,E1 -680.876,E2 -680.876} C_VEL
LIN {X 0,Y 601.437,Z 643.373,A -85,B 0,C 180,E1 -683.733,E2 -683.733} C_VEL
LIN {X 0,Y 601.426,Z 643.374,A -85,B 0,C 180,E1 -686.063,E2 -686.063} C_VEL
LIN {X 0,Y 601.432,Z 643.373,A -85,B 0,C 180,E1 -688.541,E2 -688.541} C_VEL
LIN {X 0,Y 601.433,Z 643.381,A -85,B 0,C 180,E1 -691.374,E2 -691.374} C_VEL
LIN {X 0,Y 601.413,Z 643.378,A -85,B 0,C 180,E1 -694.13,E2 -694.13} C_VEL
LIN {X 0,Y 601.415,Z 643.375,A -85,B 0,C 180,E1 -696.59,E2 -696.59} C_VEL
LIN {X 0,Y 601.425,Z 643.379,A -85,B 0,C 180,E1 -699.478,E2 -699.478} C_VEL
LIN {X 0,Y 601.398,Z 643.382,A -85,B 0,C 180,E1 -702.312,E2 -702.312} C_VEL
LIN {X 0,Y 601.415,Z 643.38,A -85,B 0,C 180,E1 -704.409,E2 -704.409} C_VEL
LIN {X 0,Y 601.414,Z 643.375,A -85,B 0,C 180,E1 -707.172,E2 -707.172} C_VEL
LIN {X 0,Y 601.435,Z 643.378,A -85,B 0,C 180,E1 -709.905,E2 -709.905} C_VEL
LIN {X 0,Y 601.445,Z 643.378,A -85,B 0,C 180,E1 -712.615,E2 -712.615} C_VEL
LIN {X 0,Y 601.427,Z 643.374,A -85,B 0,C 180,E1 -715.308,E2 -715.308} C_VEL
LIN {X 0,Y 601.417,Z 643.376,A -85,B 0,C 180,E1 -717.991,E2 -717.991} C_VEL
LIN {X 0,Y 601.454,Z 643.383,A -85,B 0,C 180,E1 -720.67,E2 -720.67} C_VEL
LIN {X 0,Y 601.426,Z 643.376,A -85,B 0,C 180,E1 -723.35,E2 -723.35} C_VEL
LIN {X 0,Y 601.43,Z 643.374,A -85,B 0,C 180,E1 -726.037,E2 -726.037} C_VEL
LIN {X 0,Y 601.43,Z 643.379,A -85,B 0,C 180,E1 -728.738,E2 -728.738} C_VEL
LIN {X 0,Y 601.43,Z 643.378,A -85,B 0,C 180,E1 -731.458,E2 -731.458} C_VEL
LIN {X 0,Y 601.408,Z 643.376,A -85,B 0,C 180,E1 -734.206,E2 -734.206} C_VEL
LIN {X 0,Y 601.426,Z 643.379,A -85,B 0,C 180,E1 -736.986,E2 -736.986} C_VEL
LIN {X 0,Y 601.406,Z 643.381,A -85,B 0,C 180,E1 -739.809,E2 -739.809} C_VEL
LIN {X 0,Y 601.409,Z 643.376,A -85,B 0,C 180,E1 -742.683,E2 -742.683} C_VEL
LIN {X 0,Y 601.398,Z 643.378,A -85,B 0,C 180,E1 -744.879,E2 -744.879} C_VEL
LIN {X 0,Y 601.418,Z 643.383,A -85,B 0,C 180,E1 -747.868,E2 -747.868} C_VEL
LIN {X 0,Y 601.439,Z 643.378,A -85,B 0,C 180,E1 -750.163,E2 -750.163} C_VEL
LIN {X 0,Y 601.416,Z 643.376,A -85,B 0,C 180,E1 -752.717,E2 -752.717} C_VEL
LIN {X 0,Y 601.412,Z 643.375,A -85,B 0,C 180,E1 -755.116,E2 -755.116} C_VEL
LIN {X 0,Y 601.429,Z 643.374,A -85,B 0,C 180,E1 -757.419,E2 -757.419} C_VEL
LIN {X 0,Y 601.412,Z 643.382,A -85,B 0,C 180,E1 -759.995,E2 -759.995} C_VEL
LIN {X 0,Y 601.434,Z 643.379,A -85,B 0,C 180,E1 -762.668,E2 -762.668} C_VEL
LIN {X 0,Y 601.418,Z 643.374,A -85,B 0,C 180,E1 -765.483,E2 -765.483} C_VEL
LIN {X 0,Y 601.421,Z 643.383,A -85,B 0,C 180,E1 -768.407,E2 -768.407} C_VEL
LIN {X 0,Y 601.431,Z 643.382,A -85,B 0,C 180,E1 -770.876,E2 -770.876} C_VEL
LIN {X 0,Y 601.439,Z 643.371,A -85,B 0,C 180,E1 -773.734,E2 -773.734} C_VEL
LIN {X 0,Y 601.425,Z 643.382,A -85,B 0,C 180,E1 -776.687,E2 -776.687} C_VEL
LIN {X 0,Y 601.433,Z 643.385,A -85,B 0,C 180,E1 -779.06,E2 -779.06} C_VEL
LIN {X 0,Y 601.46,Z 643.595,A -85,B 0,C 180,E1 -780.767,E2 -780.767} C_VEL
LIN {X 0,Y 601.993,Z 646.975,A -85,B 0,C 180,E1 -781.264,E2 -781.264} C_VEL
LIN {X 0,Y 601.877,Z 668.519,A -85,B 0,C 180,E1 -784.041,E2 -784.041} C_VEL
LIN {X 0,Y 601.741,Z 690.455,A -85,B 0,C 180,E1 -786.804,E2 -786.804} C_VEL
LIN {X 0,Y 601.772,Z 696.057,A -85,B 0,C 180,E1 -787.471,E2 -787.471} C_VEL
LIN {X 0,Y 602.34,Z 698.754,A -85,B 0,C 180,E1 -787.542,E2 -787.542} C_VEL
LIN {X 0,Y 602.127,Z 898.968,A -85,B 0,C 180,E1 -790.06,E2 -790.06} C_VEL
LIN {X 0,Y 602.072,Z 915.206,A -85,B 0,C 180,E1 -790.392,E2 -790.392} C_VEL
LIN {X 0,Y 602.005,Z 931.97,A -85,B 0,C 180,E1 -790.877,E2 -790.877} C_VEL
LIN {X 0,Y 601.913,Z 947.238,A -85,B 0,C 180,E1 -791.453,E2 -791.453} C_VEL
LIN {X 0,Y 601.844,Z 962.025,A -85,B 0,C 180,E1 -792.15,E2 -792.15} C_VEL
LIN {X 0,Y 601.754,Z 975.84,A -85,B 0,C 180,E1 -792.936,E2 -792.936} C_VEL
LIN {X 0,Y 601.695,Z 990.059,A -85,B 0,C 180,E1 -793.895,E2 -793.895} C_VEL
LIN {X 0,Y 601.592,Z 1003.132,A -85,B 0,C 180,E1 -794.934,E2 -794.934} C_VEL
LIN {X 0,Y 601.553,Z 1015.671,A -85,B 0,C 180,E1 -796.109,E2 -796.109} C_VEL
LIN {X 0,Y 601.472,Z 1026.911,A -85,B 0,C 180,E1 -797.345,E2 -797.345} C_VEL
LIN {X 0,Y 601.428,Z 1037.287,A -85,B 0,C 180,E1 -798.691,E2 -798.691} C_VEL
LIN {X 0,Y 601.381,Z 1046.277,A -85,B 0,C 180,E1 -800.074,E2 -800.074} C_VEL
LIN {X 0,Y 601.365,Z 1054.484,A -85,B 0,C 180,E1 -801.6,E2 -801.6} C_VEL
LIN {X 0,Y 601.367,Z 1060.461,A -85,B 0,C 180,E1 -802.952,E2 -802.952} C_VEL
LIN {X 0,Y 601.348,Z 1066.243,A -85,B 0,C 180,E1 -804.635,E2 -804.635} C_VEL
LIN {X 0,Y 601.339,Z 1069.636,A -85,B 0,C 180,E1 -805.979,E2 -805.979} C_VEL
LIN {X 0,Y 601.311,Z 1072.085,A -85,B 0,C 180,E1 -807.32,E2 -807.32} C_VEL
LIN {X 0,Y 601.345,Z 1073.48,A -85,B 0,C 180,E1 -808.661,E2 -808.661} C_VEL
LIN {X 0,Y 601.33,Z 1074,A -85,B 0,C 180,E1 -810,E2 -810} C_VEL
LIN {X 0,Y 601.345,Z 1073.48,A -85,B 0,C 180,E1 -811.339,E2 -811.339} C_VEL
LIN {X 0,Y 601.311,Z 1072.085,A -85,B 0,C 180,E1 -812.68,E2 -812.68} C_VEL
LIN {X 0,Y 601.339,Z 1069.636,A -85,B 0,C 180,E1 -814.021,E2 -814.021} C_VEL
LIN {X 0,Y 601.348,Z 1066.243,A -85,B 0,C 180,E1 -815.365,E2 -815.365} C_VEL
LIN {X 0,Y 601.367,Z 1060.461,A -85,B 0,C 180,E1 -817.048,E2 -817.048} C_VEL
LIN {X 0,Y 601.365,Z 1054.484,A -85,B 0,C 180,E1 -818.4,E2 -818.4} C_VEL
LIN {X 0,Y 601.381,Z 1046.277,A -85,B 0,C 180,E1 -819.926,E2 -819.926} C_VEL
LIN {X 0,Y 601.441,Z 1037.393,A -85,B 0,C 180,E1 -821.294,E2 -821.294} C_VEL
LIN {X 0,Y 601.472,Z 1026.911,A -85,B 0,C 180,E1 -822.655,E2 -822.655} C_VEL
LIN {X 0,Y 601.552,Z 1015.672,A -85,B 0,C 180,E1 -823.891,E2 -823.891} C_VEL
LIN {X 0,Y 601.593,Z 1003.132,A -85,B 0,C 180,E1 -825.066,E2 -825.066} C_VEL
LIN {X 0,Y 601.695,Z 990.059,A -85,B 0,C 180,E1 -826.105,E2 -826.105} C_VEL
LIN {X 0,Y 601.754,Z 975.84,A -85,B 0,C 180,E1 -827.064,E2 -827.064} C_VEL
LIN {X 0,Y 601.844,Z 962.025,A -85,B 0,C 180,E1 -827.85,E2 -827.85} C_VEL
LIN {X 0,Y 601.912,Z 947.238,A -85,B 0,C 180,E1 -828.547,E2 -828.547} C_VEL
LIN {X 0,Y 601.985,Z 930.677,A -85,B 0,C 180,E1 -829.168,E2 -829.168} C_VEL
LIN {X 0,Y 602.053,Z 914.293,A -85,B 0,C 180,E1 -829.631,E2 -829.631} C_VEL
LIN {X 0,Y 602.117,Z 897.471,A -85,B 0,C 180,E1 -829.962,E2 -829.962} C_VEL
LIN {X 0,Y 602.349,Z 698.799,A -85,B 0,C 180,E1 -832.457,E2 -832.457} C_VEL
LIN {X 0,Y 601.763,Z 695.783,A -85,B 0,C 180,E1 -832.546,E2 -832.546} C_VEL
LIN {X 0,Y 601.849,Z 674.276,A -85,B 0,C 180,E1 -835.227,E2 -835.227} C_VEL
LIN {X 0,Y 601.978,Z 650.956,A -85,B 0,C 180,E1 -838.217,E2 -838.217} C_VEL
LIN {X 0,Y 601.934,Z 645.937,A -85,B 0,C 180,E1 -838.875,E2 -838.875} C_VEL
LIN {X 0,Y 601.446,Z 643.461,A -85,B 0,C 180,E1 -839.273,E2 -839.273} C_VEL
LIN {X 0,Y 601.412,Z 643.376,A -85,B 0,C 180,E1 -841.725,E2 -841.725} C_VEL
LIN {X 0,Y 601.425,Z 643.375,A -85,B 0,C 180,E1 -844.118,E2 -844.118} C_VEL
LIN {X 0,Y 601.411,Z 643.376,A -85,B 0,C 180,E1 -846.581,E2 -846.581} C_VEL
LIN {X 0,Y 601.435,Z 643.38,A -85,B 0,C 180,E1 -849.535,E2 -849.535} C_VEL
LIN {X 0,Y 601.418,Z 643.38,A -85,B 0,C 180,E1 -851.764,E2 -851.764} C_VEL
LIN {X 0,Y 601.417,Z 643.374,A -85,B 0,C 180,E1 -854.535,E2 -854.535} C_VEL
LIN {X 0,Y 601.436,Z 643.38,A -85,B 0,C 180,E1 -857.405,E2 -857.405} C_VEL
LIN {X 0,Y 601.435,Z 643.374,A -85,B 0,C 180,E1 -860.463,E2 -860.463} C_VEL
LIN {X 0,Y 601.411,Z 643.379,A -85,B 0,C 180,E1 -863.418,E2 -863.418} C_VEL
LIN {X 0,Y 601.429,Z 643.384,A -85,B 0,C 180,E1 -866.063,E2 -866.063} C_VEL
LIN {X 0,Y 601.433,Z 643.376,A -85,B 0,C 180,E1 -868.541,E2 -868.541} C_VEL
LIN {X 0,Y 601.431,Z 643.371,A -85,B 0,C 180,E1 -871.373,E2 -871.373} C_VEL
LIN {X 0,Y 601.418,Z 643.383,A -85,B 0,C 180,E1 -874.129,E2 -874.129} C_VEL
LIN {X 0,Y 601.417,Z 643.383,A -85,B 0,C 180,E1 -876.59,E2 -876.59} C_VEL
LIN {X 0,Y 601.425,Z 643.374,A -85,B 0,C 180,E1 -879.478,E2 -879.478} C_VEL
LIN {X 0,Y 601.399,Z 643.383,A -85,B 0,C 180,E1 -882.312,E2 -882.312} C_VEL
LIN {X 0,Y 601.422,Z 643.38,A -85,B 0,C 180,E1 -884.409,E2 -884.409} C_VEL
LIN {X 0,Y 601.417,Z 643.38,A -85,B 0,C 180,E1 -887.172,E2 -887.172} C_VEL
LIN {X 0,Y 601.435,Z 643.373,A -85,B 0,C 180,E1 -889.905,E2 -889.905} C_VEL
LIN {X 0,Y 601.446,Z 643.374,A -85,B 0,C 180,E1 -892.615,E2 -892.615} C_VEL
LIN {X 0,Y 601.426,Z 643.383,A -85,B 0,C 180,E1 -895.308,E2 -895.308} C_VEL
LIN {X 0,Y 601.417,Z 643.376,A -85,B 0,C 180,E1 -897.991,E2 -897.991} C_VEL
LIN {X 0,Y 601.45,Z 643.372,A -85,B 0,C 180,E1 -900.669,E2 -900.669} C_VEL
LIN {X 0,Y 601.428,Z 643.382,A -85,B 0,C 180,E1 -903.349,E2 -903.349} C_VEL
LIN {X 0,Y 601.43,Z 643.377,A -85,B 0,C 180,E1 -906.037,E2 -906.037} C_VEL
LIN {X 0,Y 601.429,Z 643.373,A -85,B 0,C 180,E1 -908.737,E2 -908.737} C_VEL
LIN {X 0,Y 601.429,Z 643.379,A -85,B 0,C 180,E1 -911.458,E2 -911.458} C_VEL
LIN {X 0,Y 601.405,Z 643.378,A -85,B 0,C 180,E1 -912.383,E2 -912.383} C_VEL
LIN {X 0,Y 600.737,Z 643.462,A -85,B 0,C 180,E1 -912.942,E2 -912.942} C_VEL
LIN {X 0,Y 597.885,Z 643.825,A -85,B 0,C 180,E1 -913.85,E2 -913.85} C_VEL
LIN {X 0,Y 595.476,Z 644.119,A -85,B 0,C 180,E1 -914.58,E2 -914.58} C_VEL
LIN {X 0,Y 594.442,Z 644.245,A -85,B 0,C 180,E1 -915.143,E2 -915.143} C_VEL
LIN {X 0,Y 594.358,Z 644.256,A -85,B 0,C 180,E1 -915.334,E2 -915.334} C_VEL
LIN {X 0,Y 594.376,Z 644.26,A -85,B 0,C 180,E1 -917.904,E2 -917.904} C_VEL
LIN {X 0,Y 594.372,Z 644.253,A -85,B 0,C 180,E1 -920.918,E2 -920.918} C_VEL
LIN {X 0,Y 594.384,Z 644.253,A -85,B 0,C 180,E1 -923.704,E2 -923.704} C_VEL
LIN {X 0,Y 594.379,Z 644.257,A -85,B 0,C 180,E1 -926.699,E2 -926.699} C_VEL
LIN {X 0,Y 594.378,Z 644.253,A -85,B 0,C 180,E1 -928.998,E2 -928.998} C_VEL
LIN {X 0,Y 594.383,Z 644.251,A -85,B 0,C 180,E1 -931.646,E2 -931.646} C_VEL
LIN {X 0,Y 594.392,Z 644.258,A -85,B 0,C 180,E1 -934.579,E2 -934.579} C_VEL
LIN {X 0,Y 594.379,Z 644.259,A -85,B 0,C 180,E1 -937.087,E2 -937.087} C_VEL
LIN {X 0,Y 594.372,Z 644.253,A -85,B 0,C 180,E1 -939.776,E2 -939.776} C_VEL
LIN {X 0,Y 594.379,Z 644.253,A -85,B 0,C 180,E1 -942.374,E2 -942.374} C_VEL
LIN {X 0,Y 594.354,Z 644.267,A -85,B 0,C 180,E1 -945.192,E2 -945.192} C_VEL
LIN {X 0,Y 594.361,Z 644.26,A -85,B 0,C 180,E1 -947.625,E2 -947.625} C_VEL
LIN {X 0,Y 594.385,Z 644.251,A -85,B 0,C 180,E1 -950.322,E2 -950.322} C_VEL
LIN {X 0,Y 594.378,Z 644.254,A -85,B 0,C 180,E1 -952.914,E2 -952.914} C_VEL
LIN {X 0,Y 594.377,Z 644.259,A -85,B 0,C 180,E1 -955.861,E2 -955.861} C_VEL
LIN {X 0,Y 594.386,Z 644.251,A -85,B 0,C 180,E1 -958.652,E2 -958.652} C_VEL
LIN {X 0,Y 594.376,Z 644.253,A -85,B 0,C 180,E1 -961.042,E2 -961.042} C_VEL
LIN {X 0,Y 594.384,Z 644.253,A -85,B 0,C 180,E1 -963.301,E2 -963.301} C_VEL
LIN {X 0,Y 594.388,Z 644.258,A -85,B 0,C 180,E1 -966.297,E2 -966.297} C_VEL
LIN {X 0,Y 594.402,Z 644.249,A -85,B 0,C 180,E1 -969.225,E2 -969.225} C_VEL
LIN {X 0,Y 594.35,Z 644.264,A -85,B 0,C 180,E1 -972.095,E2 -972.095} C_VEL
LIN {X 0,Y 594.362,Z 644.263,A -85,B 0,C 180,E1 -974.219,E2 -974.219} C_VEL
LIN {X 0,Y 594.363,Z 644.257,A -85,B 0,C 180,E1 -977.017,E2 -977.017} C_VEL
LIN {X 0,Y 594.388,Z 644.252,A -85,B 0,C 180,E1 -979.784,E2 -979.784} C_VEL
LIN {X 0,Y 594.39,Z 644.259,A -85,B 0,C 180,E1 -982.527,E2 -982.527} C_VEL
LIN {X 0,Y 594.386,Z 644.255,A -85,B 0,C 180,E1 -985.252,E2 -985.252} C_VEL
LIN {X 0,Y 594.398,Z 644.25,A -85,B 0,C 180,E1 -987.967,E2 -987.967} C_VEL
LIN {X 0,Y 594.414,Z 644.253,A -85,B 0,C 180,E1 -990.677,E2 -990.677} C_VEL
LIN {X 0,Y 594.383,Z 644.259,A -85,B 0,C 180,E1 -993.389,E2 -993.389} C_VEL
LIN {X 0,Y 594.363,Z 644.255,A -85,B 0,C 180,E1 -996.109,E2 -996.109} C_VEL
LIN {X 0,Y 594.395,Z 644.253,A -85,B 0,C 180,E1 -998.842,E2 -998.842} C_VEL
LIN {X 0,Y 594.389,Z 644.26,A -85,B 0,C 180,E1 -1001.595,E2 -1001.595} C_VEL
LIN {X 0,Y 594.385,Z 644.252,A -85,B 0,C 180,E1 -1004.377,E2 -1004.377} C_VEL
LIN {X 0,Y 594.386,Z 644.254,A -85,B 0,C 180,E1 -1007.193,E2 -1007.193} C_VEL
LIN {X 0,Y 594.371,Z 644.26,A -85,B 0,C 180,E1 -1010.053,E2 -1010.053} C_VEL
LIN {X 0,Y 594.36,Z 644.255,A -85,B 0,C 180,E1 -1012.967,E2 -1012.967} C_VEL
LIN {X 0,Y 594.37,Z 644.254,A -85,B 0,C 180,E1 -1015.193,E2 -1015.193} C_VEL
LIN {X 0,Y 594.379,Z 644.254,A -85,B 0,C 180,E1 -1017.526,E2 -1017.526} C_VEL
LIN {X 0,Y 594.39,Z 644.256,A -85,B 0,C 180,E1 -1020.558,E2 -1020.558} C_VEL
LIN {X 0,Y 594.373,Z 644.255,A -85,B 0,C 180,E1 -1022.949,E2 -1022.949} C_VEL
LIN {X 0,Y 594.374,Z 644.253,A -85,B 0,C 180,E1 -1025.406,E2 -1025.406} C_VEL
LIN {X 0,Y 594.377,Z 644.254,A -85,B 0,C 180,E1 -1027.94,E2 -1027.94} C_VEL
LIN {X 0,Y 594.373,Z 644.261,A -85,B 0,C 180,E1 -1030.822,E2 -1030.822} C_VEL
LIN {X 0,Y 594.372,Z 644.253,A -85,B 0,C 180,E1 -1033.841,E2 -1033.841} C_VEL
LIN {X 0,Y 594.377,Z 644.26,A -85,B 0,C 180,E1 -1036.702,E2 -1036.702} C_VEL
LIN {X 0,Y 594.382,Z 644.256,A -85,B 0,C 180,E1 -1039.435,E2 -1039.435} C_VEL
LIN {X 0,Y 594.382,Z 644.252,A -85,B 0,C 180,E1 -1042.391,E2 -1042.391} C_VEL
LIN {X 0,Y 594.378,Z 644.252,A -85,B 0,C 180,E1 -1044.671,E2 -1044.671} C_VEL
LIN {X 0,Y 594.369,Z 644.26,A -85,B 0,C 180,E1 -1047.088,E2 -1047.088} C_VEL
LIN {X 0,Y 594.389,Z 644.255,A -85,B 0,C 180,E1 -1049.669,E2 -1049.669} C_VEL
LIN {X 0,Y 594.361,Z 644.252,A -85,B 0,C 180,E1 -1052.539,E2 -1052.539} C_VEL
LIN {X 0,Y 594.372,Z 644.253,A -85,B 0,C 180,E1 -1054.807,E2 -1054.807} C_VEL
LIN {X 0,Y 594.393,Z 644.253,A -85,B 0,C 180,E1 -1057.255,E2 -1057.255} C_VEL
LIN {X 0,Y 594.373,Z 644.262,A -85,B 0,C 180,E1 -1059.947,E2 -1059.947} C_VEL
LIN {X 0,Y 594.383,Z 644.251,A -85,B 0,C 180,E1 -1062.807,E2 -1062.807} C_VEL
LIN {X 0,Y 594.378,Z 644.259,A -85,B 0,C 180,E1 -1065.825,E2 -1065.825} C_VEL
LIN {X 0,Y 594.387,Z 644.258,A -85,B 0,C 180,E1 -1068.404,E2 -1068.404} C_VEL
LIN {X 0,Y 594.391,Z 644.25,A -85,B 0,C 180,E1 -1071.158,E2 -1071.158} C_VEL
LIN {X 0,Y 594.383,Z 644.254,A -85,B 0,C 180,E1 -1073.891,E2 -1073.891} C_VEL
LIN {X 0,Y 594.379,Z 644.26,A -85,B 0,C 180,E1 -1076.611,E2 -1076.611} C_VEL
LIN {X 0,Y 594.42,Z 644.248,A -85,B 0,C 180,E1 -1079.323,E2 -1079.323} C_VEL
LIN {X 0,Y 594.388,Z 644.251,A -85,B 0,C 180,E1 -1082.033,E2 -1082.033} C_VEL
LIN {X 0,Y 594.394,Z 644.26,A -85,B 0,C 180,E1 -1084.748,E2 -1084.748} C_VEL
LIN {X 0,Y 594.41,Z 644.249,A -85,B 0,C 180,E1 -1087.473,E2 -1087.473} C_VEL
LIN {X 0,Y 594.393,Z 644.25,A -85,B 0,C 180,E1 -1090.216,E2 -1090.216} C_VEL
LIN {X 0,Y 594.366,Z 644.261,A -85,B 0,C 180,E1 -1092.983,E2 -1092.983} C_VEL
LIN {X 0,Y 594.368,Z 644.256,A -85,B 0,C 180,E1 -1095.781,E2 -1095.781} C_VEL
LIN {X 0,Y 594.377,Z 644.252,A -85,B 0,C 180,E1 -1098.618,E2 -1098.618} C_VEL
LIN {X 0,Y 594.362,Z 644.265,A -85,B 0,C 180,E1 -1101.504,E2 -1101.504} C_VEL
LIN {X 0,Y 594.378,Z 644.253,A -85,B 0,C 180,E1 -1104.447,E2 -1104.447} C_VEL
LIN {X 0,Y 594.38,Z 644.251,A -85,B 0,C 180,E1 -1106.7,E2 -1106.7} C_VEL
LIN {X 0,Y 594.378,Z 644.248,A -85,B 0,C 180,E1 -1108.999,E2 -1108.999} C_VEL
LIN {X 0,Y 594.385,Z 644.257,A -85,B 0,C 180,E1 -1111.646,E2 -1111.646} C_VEL
LIN {X 0,Y 594.394,Z 644.251,A -85,B 0,C 180,E1 -1114.579,E2 -1114.579} C_VEL
LIN {X 0,Y 594.381,Z 644.251,A -85,B 0,C 180,E1 -1117.087,E2 -1117.087} C_VEL
LIN {X 0,Y 594.374,Z 644.256,A -85,B 0,C 180,E1 -1119.776,E2 -1119.776} C_VEL
LIN {X 0,Y 594.384,Z 644.262,A -85,B 0,C 180,E1 -1122.374,E2 -1122.374} C_VEL
LIN {X 0,Y 594.356,Z 644.254,A -85,B 0,C 180,E1 -1125.192,E2 -1125.192} C_VEL
LIN {X 0,Y 594.363,Z 644.254,A -85,B 0,C 180,E1 -1127.626,E2 -1127.626} C_VEL
LIN {X 0,Y 594.387,Z 644.256,A -85,B 0,C 180,E1 -1130.322,E2 -1130.322} C_VEL
LIN {X 0,Y 594.383,Z 644.256,A -85,B 0,C 180,E1 -1132.914,E2 -1132.914} C_VEL
LIN {X 0,Y 594.379,Z 644.253,A -85,B 0,C 180,E1 -1135.862,E2 -1135.862} C_VEL
LIN {X 0,Y 594.389,Z 644.254,A -85,B 0,C 180,E1 -1138.652,E2 -1138.652} C_VEL
LIN {X 0,Y 594.412,Z 644.434,A -85,B 0,C 180,E1 -1140.495,E2 -1140.495} C_VEL
LIN {X 0,Y 595.204,Z 648.041,A -85,B 0,C 180,E1 -1141.046,E2 -1141.046} C_VEL
LIN {X 0,Y 595.085,Z 667.979,A -85,B 0,C 180,E1 -1143.653,E2 -1143.653} C_VEL
LIN {X 0,Y 594.914,Z 690.309,A -85,B 0,C 180,E1 -1146.503,E2 -1146.503} C_VEL
LIN {X 0,Y 594.925,Z 696.164,A -85,B 0,C 180,E1 -1147.203,E2 -1147.203} C_VEL
LIN {X 0,Y 595.805,Z 700.196,A -85,B 0,C 180,E1 -1147.3,E2 -1147.3} C_VEL
LIN {X 0,Y 595.474,Z 898.928,A -85,B 0,C 180,E1 -1149.828,E2 -1149.828} C_VEL
LIN {X 0,Y 595.353,Z 915.212,A -85,B 0,C 180,E1 -1150.161,E2 -1150.161} C_VEL
LIN {X 0,Y 595.265,Z 931.98,A -85,B 0,C 180,E1 -1150.652,E2 -1150.652} C_VEL
LIN {X 0,Y 595.145,Z 947.472,A -85,B 0,C 180,E1 -1151.245,E2 -1151.245} C_VEL
LIN {X 0,Y 595.041,Z 962.027,A -85,B 0,C 180,E1 -1151.939,E2 -1151.939} C_VEL
LIN {X 0,Y 594.894,Z 975.838,A -85,B 0,C 180,E1 -1152.734,E2 -1152.734} C_VEL
LIN {X 0,Y 594.801,Z 990.065,A -85,B 0,C 180,E1 -1153.703,E2 -1153.703} C_VEL
LIN {X 0,Y 594.647,Z 1003.132,A -85,B 0,C 180,E1 -1154.754,E2 -1154.754} C_VEL
LIN {X 0,Y 594.557,Z 1015.304,A -85,B 0,C 180,E1 -1155.904,E2 -1155.904} C_VEL
LIN {X 0,Y 594.449,Z 1026.904,A -85,B 0,C 180,E1 -1157.193,E2 -1157.193} C_VEL
LIN {X 0,Y 594.381,Z 1037.423,A -85,B 0,C 180,E1 -1158.574,E2 -1158.574} C_VEL
LIN {X 0,Y 594.329,Z 1046.28,A -85,B 0,C 180,E1 -1159.955,E2 -1159.955} C_VEL
LIN {X 0,Y 594.295,Z 1054.482,A -85,B 0,C 180,E1 -1161.499,E2 -1161.499} C_VEL
LIN {X 0,Y 594.29,Z 1060.455,A -85,B 0,C 180,E1 -1162.867,E2 -1162.867} C_VEL
LIN {X 0,Y 594.265,Z 1066.241,A -85,B 0,C 180,E1 -1164.571,E2 -1164.571} C_VEL
LIN {X 0,Y 594.251,Z 1069.639,A -85,B 0,C 180,E1 -1165.931,E2 -1165.931} C_VEL
LIN {X 0,Y 594.213,Z 1072.085,A -85,B 0,C 180,E1 -1167.288,E2 -1167.288} C_VEL
LIN {X 0,Y 594.244,Z 1073.483,A -85,B 0,C 180,E1 -1168.645,E2 -1168.645} C_VEL
LIN {X 0,Y 594.231,Z 1074,A -85,B 0,C 180,E1 -1170,E2 -1170} C_VEL
LIN {X 0,Y 594.244,Z 1073.483,A -85,B 0,C 180,E1 -1171.355,E2 -1171.355} C_VEL
LIN {X 0,Y 594.213,Z 1072.085,A -85,B 0,C 180,E1 -1172.712,E2 -1172.712} C_VEL
LIN {X 0,Y 594.251,Z 1069.639,A -85,B 0,C 180,E1 -1174.069,E2 -1174.069} C_VEL
LIN {X 0,Y 594.277,Z 1065.18,A -85,B 0,C 180,E1 -1175.769,E2 -1175.769} C_VEL
LIN {X 0,Y 594.29,Z 1060.455,A -85,B 0,C 180,E1 -1177.133,E2 -1177.133} C_VEL
LIN {X 0,Y 594.295,Z 1054.482,A -85,B 0,C 180,E1 -1178.501,E2 -1178.501} C_VEL
LIN {X 0,Y 594.329,Z 1046.28,A -85,B 0,C 180,E1 -1180.045,E2 -1180.045} C_VEL
LIN {X 0,Y 594.406,Z 1037.543,A -85,B 0,C 180,E1 -1181.409,E2 -1181.409} C_VEL
LIN {X 0,Y 594.461,Z 1028.342,A -85,B 0,C 180,E1 -1182.633,E2 -1182.633} C_VEL
LIN {X 0,Y 594.551,Z 1016.978,A -85,B 0,C 180,E1 -1183.92,E2 -1183.92} C_VEL
LIN {X 0,Y 594.637,Z 1005.072,A -85,B 0,C 180,E1 -1185.071,E2 -1185.071} C_VEL
LIN {X 0,Y 594.787,Z 991.226,A -85,B 0,C 180,E1 -1186.209,E2 -1186.209} C_VEL
LIN {X 0,Y 594.9,Z 977.249,A -85,B 0,C 180,E1 -1187.178,E2 -1187.178} C_VEL
LIN {X 0,Y 595.029,Z 963.699,A -85,B 0,C 180,E1 -1187.972,E2 -1187.972} C_VEL
LIN {X 0,Y 595.129,Z 948.669,A -85,B 0,C 180,E1 -1188.701,E2 -1188.701} C_VEL
LIN {X 0,Y 595.281,Z 933.273,A -85,B 0,C 180,E1 -1189.303,E2 -1189.303} C_VEL
LIN {X 0,Y 595.358,Z 917.038,A -85,B 0,C 180,E1 -1189.794,E2 -1189.794} C_VEL
LIN {X 0,Y 595.439,Z 900.333,A -85,B 0,C 180,E1 -1190.151,E2 -1190.151} C_VEL
LIN {X 0,Y 595.57,Z 830.152,A -85,B 0,C 180,E1 -1191.055,E2 -1191.055} C_VEL
LIN {X 0,Y 595.733,Z 699.559,A -85,B 0,C 180,E1 -1192.711,E2 -1192.711} C_VEL
LIN {X 0,Y 594.89,Z 695.731,A -85,B 0,C 180,E1 -1192.825,E2 -1192.825} C_VEL
LIN {X 0,Y 595.019,Z 674.276,A -85,B 0,C 180,E1 -1195.538,E2 -1195.538} C_VEL
LIN {X 0,Y 595.215,Z 652.413,A -85,B 0,C 180,E1 -1198.375,E2 -1198.375} C_VEL
LIN {X 0,Y 595.068,Z 647.167,A -85,B 0,C 180,E1 -1199.077,E2 -1199.077} C_VEL
LIN {X 0,Y 594.406,Z 644.341,A -85,B 0,C 180,E1 -1199.53,E2 -1199.53} C_VEL
LIN {X 0,Y 594.371,Z 644.252,A -85,B 0,C 180,E1 -1202.146,E2 -1202.146} C_VEL
LIN {X 0,Y 594.391,Z 644.254,A -85,B 0,C 180,E1 -1204.578,E2 -1204.578} C_VEL
LIN {X 0,Y 594.383,Z 644.256,A -85,B 0,C 180,E1 -1207.086,E2 -1207.086} C_VEL
LIN {X 0,Y 594.37,Z 644.257,A -85,B 0,C 180,E1 -1209.774,E2 -1209.774} C_VEL
LIN {X 0,Y 594.363,Z 644.254,A -85,B 0,C 180,E1 -1212.374,E2 -1212.374} C_VEL
LIN {X 0,Y 594.355,Z 644.258,A -85,B 0,C 180,E1 -1215.191,E2 -1215.191} C_VEL
LIN {X 0,Y 594.384,Z 644.262,A -85,B 0,C 180,E1 -1217.626,E2 -1217.626} C_VEL
LIN {X 0,Y 594.389,Z 644.253,A -85,B 0,C 180,E1 -1220.321,E2 -1220.321} C_VEL
LIN {X 0,Y 594.381,Z 644.251,A -85,B 0,C 180,E1 -1222.913,E2 -1222.913} C_VEL
LIN {X 0,Y 594.382,Z 644.26,A -85,B 0,C 180,E1 -1225.859,E2 -1225.859} C_VEL
LIN {X 0,Y 594.382,Z 644.253,A -85,B 0,C 180,E1 -1228.65,E2 -1228.65} C_VEL
LIN {X 0,Y 594.38,Z 644.248,A -85,B 0,C 180,E1 -1231.04,E2 -1231.04} C_VEL
LIN {X 0,Y 594.39,Z 644.255,A -85,B 0,C 180,E1 -1233.973,E2 -1233.973} C_VEL
LIN {X 0,Y 594.387,Z 644.261,A -85,B 0,C 180,E1 -1236.296,E2 -1236.296} C_VEL
LIN {X 0,Y 594.396,Z 644.251,A -85,B 0,C 180,E1 -1239.224,E2 -1239.224} C_VEL
LIN {X 0,Y 594.376,Z 644.254,A -85,B 0,C 180,E1 -1242.096,E2 -1242.096} C_VEL
LIN {X 0,Y 594.375,Z 644.255,A -85,B 0,C 180,E1 -1244.219,E2 -1244.219} C_VEL
LIN {X 0,Y 594.366,Z 644.261,A -85,B 0,C 180,E1 -1247.017,E2 -1247.017} C_VEL
LIN {X 0,Y 594.393,Z 644.25,A -85,B 0,C 180,E1 -1249.784,E2 -1249.784} C_VEL
LIN {X 0,Y 594.41,Z 644.249,A -85,B 0,C 180,E1 -1252.527,E2 -1252.527} C_VEL
LIN {X 0,Y 594.394,Z 644.259,A -85,B 0,C 180,E1 -1255.252,E2 -1255.252} C_VEL
LIN {X 0,Y 594.388,Z 644.251,A -85,B 0,C 180,E1 -1257.967,E2 -1257.967} C_VEL
LIN {X 0,Y 594.42,Z 644.248,A -85,B 0,C 180,E1 -1260.677,E2 -1260.677} C_VEL
LIN {X 0,Y 594.379,Z 644.26,A -85,B 0,C 180,E1 -1263.389,E2 -1263.389} C_VEL
LIN {X 0,Y 594.383,Z 644.254,A -85,B 0,C 180,E1 -1266.109,E2 -1266.109} C_VEL
LIN {X 0,Y 594.391,Z 644.25,A -85,B 0,C 180,E1 -1268.842,E2 -1268.842} C_VEL
LIN {X 0,Y 594.387,Z 644.258,A -85,B 0,C 180,E1 -1271.596,E2 -1271.596} C_VEL
LIN {X 0,Y 594.378,Z 644.256,A -85,B 0,C 180,E1 -1274.377,E2 -1274.377} C_VEL
LIN {X 0,Y 594.358,Z 644.256,A -85,B 0,C 180,E1 -1275.334,E2 -1275.334} C_VEL
LIN {X 0,Y 593.691,Z 644.347,A -85,B 0,C 180,E1 -1275.9,E2 -1275.9} C_VEL
LIN {X 0,Y 590.838,Z 644.707,A -85,B 0,C 180,E1 -1276.818,E2 -1276.818} C_VEL
LIN {X 0,Y 588.431,Z 645.008,A -85,B 0,C 180,E1 -1277.557,E2 -1277.557} C_VEL
LIN {X 0,Y 587.4,Z 645.132,A -85,B 0,C 180,E1 -1278.127,E2 -1278.127} C_VEL
LIN {X 0,Y 587.318,Z 645.138,A -85,B 0,C 180,E1 -1278.32,E2 -1278.32} C_VEL
LIN {X 0,Y 587.346,Z 645.128,A -85,B 0,C 180,E1 -1281.045,E2 -1281.045} C_VEL
LIN {X 0,Y 587.356,Z 645.126,A -85,B 0,C 180,E1 -1283.257,E2 -1283.257} C_VEL
LIN {X 0,Y 587.354,Z 645.136,A -85,B 0,C 180,E1 -1286.277,E2 -1286.277} C_VEL
LIN {X 0,Y 587.345,Z 645.127,A -85,B 0,C 180,E1 -1289.135,E2 -1289.135} C_VEL
LIN {X 0,Y 587.347,Z 645.128,A -85,B 0,C 180,E1 -1291.838,E2 -1291.838} C_VEL
LIN {X 0,Y 587.35,Z 645.132,A -85,B 0,C 180,E1 -1294.35,E2 -1294.35} C_VEL
LIN {X 0,Y 587.344,Z 645.134,A -85,B 0,C 180,E1 -1296.747,E2 -1296.747} C_VEL
LIN {X 0,Y 587.341,Z 645.133,A -85,B 0,C 180,E1 -1299.359,E2 -1299.359} C_VEL
LIN {X 0,Y 587.357,Z 645.127,A -85,B 0,C 180,E1 -1302.112,E2 -1302.112} C_VEL
LIN {X 0,Y 587.307,Z 645.143,A -85,B 0,C 180,E1 -1305.089,E2 -1305.089} C_VEL
LIN {X 0,Y 587.344,Z 645.13,A -85,B 0,C 180,E1 -1307.928,E2 -1307.928} C_VEL
LIN {X 0,Y 587.325,Z 645.136,A -85,B 0,C 180,E1 -1311.059,E2 -1311.059} C_VEL
LIN {X 0,Y 587.346,Z 645.136,A -85,B 0,C 180,E1 -1313.292,E2 -1313.292} C_VEL
LIN {X 0,Y 587.359,Z 645.135,A -85,B 0,C 180,E1 -1315.781,E2 -1315.781} C_VEL
LIN {X 0,Y 587.348,Z 645.131,A -85,B 0,C 180,E1 -1318.232,E2 -1318.232} C_VEL
LIN {X 0,Y 587.343,Z 645.129,A -85,B 0,C 180,E1 -1320.867,E2 -1320.867} C_VEL
LIN {X 0,Y 587.353,Z 645.137,A -85,B 0,C 180,E1 -1323.819,E2 -1323.819} C_VEL
LIN {X 0,Y 587.335,Z 645.141,A -85,B 0,C 180,E1 -1325.994,E2 -1325.994} C_VEL
LIN {X 0,Y 587.317,Z 645.142,A -85,B 0,C 180,E1 -1328.226,E2 -1328.226} C_VEL
LIN {X 0,Y 587.346,Z 645.129,A -85,B 0,C 180,E1 -1331.152,E2 -1331.152} C_VEL
LIN {X 0,Y 587.32,Z 645.137,A -85,B 0,C 180,E1 -1334.025,E2 -1334.025} C_VEL
LIN {X 0,Y 587.354,Z 645.134,A -85,B 0,C 180,E1 -1336.155,E2 -1336.155} C_VEL
LIN {X 0,Y 587.338,Z 645.134,A -85,B 0,C 180,E1 -1338.963,E2 -1338.963} C_VEL
LIN {X 0,Y 587.365,Z 645.126,A -85,B 0,C 180,E1 -1341.745,E2 -1341.745} C_VEL
LIN {X 0,Y 587.358,Z 645.134,A -85,B 0,C 180,E1 -1344.507,E2 -1344.507} C_VEL
LIN {X 0,Y 587.367,Z 645.131,A -85,B 0,C 180,E1 -1347.257,E2 -1347.257} C_VEL
LIN {X 0,Y 587.381,Z 645.124,A -85,B 0,C 180,E1 -1350,E2 -1350} C_VEL
LIN {X 0,Y 587.367,Z 645.131,A -85,B 0,C 180,E1 -1352.743,E2 -1352.743} C_VEL
LIN {X 0,Y 587.358,Z 645.134,A -85,B 0,C 180,E1 -1355.493,E2 -1355.493} C_VEL
LIN {X 0,Y 587.365,Z 645.126,A -85,B 0,C 180,E1 -1358.255,E2 -1358.255} C_VEL
LIN {X 0,Y 587.344,Z 645.135,A -85,B 0,C 180,E1 -1361.133,E2 -1361.133} C_VEL
LIN {X 0,Y 587.36,Z 645.128,A -85,B 0,C 180,E1 -1364.26,E2 -1364.26} C_VEL
LIN {X 0,Y 587.346,Z 645.134,A -85,B 0,C 180,E1 -1367.406,E2 -1367.406} C_VEL
LIN {X 0,Y 587.326,Z 645.134,A -85,B 0,C 180,E1 -1370.304,E2 -1370.304} C_VEL
LIN {X 0,Y 587.319,Z 645.133,A -85,B 0,C 180,E1 -1373.258,E2 -1373.258} C_VEL
LIN {X 0,Y 587.328,Z 645.134,A -85,B 0,C 180,E1 -1375.516,E2 -1375.516} C_VEL
LIN {X 0,Y 587.343,Z 645.135,A -85,B 0,C 180,E1 -1377.817,E2 -1377.817} C_VEL
LIN {X 0,Y 587.346,Z 645.135,A -85,B 0,C 180,E1 -1380.512,E2 -1380.512} C_VEL
LIN {X 0,Y 587.329,Z 645.131,A -85,B 0,C 180,E1 -1383.396,E2 -1383.396} C_VEL
LIN {X 0,Y 587.348,Z 645.13,A -85,B 0,C 180,E1 -1385.895,E2 -1385.895} C_VEL
LIN {X 0,Y 587.323,Z 645.142,A -85,B 0,C 180,E1 -1388.479,E2 -1388.479} C_VEL
LIN {X 0,Y 587.329,Z 645.134,A -85,B 0,C 180,E1 -1391.156,E2 -1391.156} C_VEL
LIN {X 0,Y 587.324,Z 645.132,A -85,B 0,C 180,E1 -1394.114,E2 -1394.114} C_VEL
LIN {X 0,Y 587.327,Z 645.141,A -85,B 0,C 180,E1 -1396.995,E2 -1396.995} C_VEL
LIN {X 0,Y 587.321,Z 645.132,A -85,B 0,C 180,E1 -1399.747,E2 -1399.747} C_VEL
LIN {X 0,Y 587.337,Z 645.129,A -85,B 0,C 180,E1 -1402.392,E2 -1402.392} C_VEL
LIN {X 0,Y 587.344,Z 645.131,A -85,B 0,C 180,E1 -1404.946,E2 -1404.946} C_VEL
LIN {X 0,Y 587.332,Z 645.14,A -85,B 0,C 180,E1 -1407.421,E2 -1407.421} C_VEL
LIN {X 0,Y 587.337,Z 645.13,A -85,B 0,C 180,E1 -1409.83,E2 -1409.83} C_VEL
LIN {X 0,Y 587.34,Z 645.127,A -85,B 0,C 180,E1 -1412.306,E2 -1412.306} C_VEL
LIN {X 0,Y 587.332,Z 645.13,A -85,B 0,C 180,E1 -1414.484,E2 -1414.484} C_VEL
LIN {X 0,Y 587.359,Z 645.133,A -85,B 0,C 180,E1 -1417.487,E2 -1417.487} C_VEL
LIN {X 0,Y 587.337,Z 645.131,A -85,B 0,C 180,E1 -1420.425,E2 -1420.425} C_VEL
LIN {X 0,Y 587.342,Z 645.129,A -85,B 0,C 180,E1 -1423.311,E2 -1423.311} C_VEL
LIN {X 0,Y 587.352,Z 645.136,A -85,B 0,C 180,E1 -1426.154,E2 -1426.154} C_VEL
LIN {X 0,Y 587.334,Z 645.13,A -85,B 0,C 180,E1 -1428.963,E2 -1428.963} C_VEL
LIN {X 0,Y 587.363,Z 645.127,A -85,B 0,C 180,E1 -1431.745,E2 -1431.745} C_VEL
LIN {X 0,Y 587.358,Z 645.137,A -85,B 0,C 180,E1 -1434.507,E2 -1434.507} C_VEL
LIN {X 0,Y 587.374,Z 645.124,A -85,B 0,C 180,E1 -1437.257,E2 -1437.257} C_VEL
LIN {X 0,Y 587.371,Z 645.126,A -85,B 0,C 180,E1 -1440,E2 -1440} C_VEL
LIN {X 0,Y 587.375,Z 645.134,A -85,B 0,C 180,E1 -1442.743,E2 -1442.743} C_VEL
LIN {X 0,Y 587.358,Z 645.128,A -85,B 0,C 180,E1 -1445.493,E2 -1445.493} C_VEL
LIN {X 0,Y 587.363,Z 645.125,A -85,B 0,C 180,E1 -1448.255,E2 -1448.255} C_VEL
LIN {X 0,Y 587.35,Z 645.138,A -85,B 0,C 180,E1 -1451.142,E2 -1451.142} C_VEL
LIN {X 0,Y 587.354,Z 645.127,A -85,B 0,C 180,E1 -1454.262,E2 -1454.262} C_VEL
LIN {X 0,Y 587.351,Z 645.137,A -85,B 0,C 180,E1 -1457.406,E2 -1457.406} C_VEL
LIN {X 0,Y 587.325,Z 645.131,A -85,B 0,C 180,E1 -1460.305,E2 -1460.305} C_VEL
LIN {X 0,Y 587.317,Z 645.136,A -85,B 0,C 180,E1 -1463.259,E2 -1463.259} C_VEL
LIN {X 0,Y 587.356,Z 645.129,A -85,B 0,C 180,E1 -1466.183,E2 -1466.183} C_VEL
LIN {X 0,Y 587.346,Z 645.124,A -85,B 0,C 180,E1 -1469.135,E2 -1469.135} C_VEL
LIN {X 0,Y 587.348,Z 645.137,A -85,B 0,C 180,E1 -1471.839,E2 -1471.839} C_VEL
LIN {X 0,Y 587.353,Z 645.131,A -85,B 0,C 180,E1 -1474.351,E2 -1474.351} C_VEL
LIN {X 0,Y 587.346,Z 645.129,A -85,B 0,C 180,E1 -1476.747,E2 -1476.747} C_VEL
LIN {X 0,Y 587.342,Z 645.129,A -85,B 0,C 180,E1 -1479.36,E2 -1479.36} C_VEL
LIN {X 0,Y 587.359,Z 645.131,A -85,B 0,C 180,E1 -1482.112,E2 -1482.112} C_VEL
LIN {X 0,Y 587.308,Z 645.133,A -85,B 0,C 180,E1 -1485.089,E2 -1485.089} C_VEL
LIN {X 0,Y 587.346,Z 645.13,A -85,B 0,C 180,E1 -1487.928,E2 -1487.928} C_VEL
LIN {X 0,Y 587.329,Z 645.135,A -85,B 0,C 180,E1 -1491.059,E2 -1491.059} C_VEL
LIN {X 0,Y 587.349,Z 645.127,A -85,B 0,C 180,E1 -1493.292,E2 -1493.292} C_VEL
LIN {X 0,Y 587.362,Z 645.128,A -85,B 0,C 180,E1 -1495.781,E2 -1495.781} C_VEL
LIN {X 0,Y 587.351,Z 645.126,A -85,B 0,C 180,E1 -1498.233,E2 -1498.233} C_VEL
LIN {X 0,Y 587.38,Z 645.327,A -85,B 0,C 180,E1 -1500.229,E2 -1500.229} C_VEL
LIN {X 0,Y 588.392,Z 649.601,A -85,B 0,C 180,E1 -1500.888,E2 -1500.888} C_VEL
LIN {X 0,Y 588.349,Z 664.074,A -85,B 0,C 180,E1 -1502.813,E2 -1502.813} C_VEL
LIN {X 0,Y 588.114,Z 685.937,A -85,B 0,C 180,E1 -1505.653,E2 -1505.653} C_VEL
LIN {X 0,Y 588.091,Z 695.964,A -85,B 0,C 180,E1 -1506.913,E2 -1506.913} C_VEL
LIN {X 0,Y 589.223,Z 700.957,A -85,B 0,C 180,E1 -1507.042,E2 -1507.042} C_VEL
LIN {X 0,Y 588.804,Z 898.889,A -85,B 0,C 180,E1 -1509.589,E2 -1509.589} C_VEL
LIN {X 0,Y 588.674,Z 915.219,A -85,B 0,C 180,E1 -1509.926,E2 -1509.926} C_VEL
LIN {X 0,Y 588.542,Z 931.99,A -85,B 0,C 180,E1 -1510.422,E2 -1510.422} C_VEL
LIN {X 0,Y 588.376,Z 947.701,A -85,B 0,C 180,E1 -1511.032,E2 -1511.032} C_VEL
LIN {X 0,Y 588.233,Z 962.015,A -85,B 0,C 180,E1 -1511.723,E2 -1511.723} C_VEL
LIN {X 0,Y 588.063,Z 975.836,A -85,B 0,C 180,E1 -1512.527,E2 -1512.527} C_VEL
LIN {X 0,Y 587.873,Z 990.07,A -85,B 0,C 180,E1 -1513.506,E2 -1513.506} C_VEL
LIN {X 0,Y 587.729,Z 1003.133,A -85,B 0,C 180,E1 -1514.57,E2 -1514.57} C_VEL
LIN {X 0,Y 587.561,Z 1015.915,A -85,B 0,C 180,E1 -1515.799,E2 -1515.799} C_VEL
LIN {X 0,Y 587.449,Z 1026.897,A -85,B 0,C 180,E1 -1517.038,E2 -1517.038} C_VEL
LIN {X 0,Y 587.349,Z 1036.209,A -85,B 0,C 180,E1 -1518.264,E2 -1518.264} C_VEL
LIN {X 0,Y 587.3,Z 1045.271,A -85,B 0,C 180,E1 -1519.66,E2 -1519.66} C_VEL
LIN {X 0,Y 587.248,Z 1052.858,A -85,B 0,C 180,E1 -1521.05,E2 -1521.05} C_VEL
LIN {X 0,Y 587.202,Z 1059.058,A -85,B 0,C 180,E1 -1522.435,E2 -1522.435} C_VEL
LIN {X 0,Y 587.162,Z 1064.115,A -85,B 0,C 180,E1 -1523.816,E2 -1523.816} C_VEL
LIN {X 0,Y 587.131,Z 1068.061,A -85,B 0,C 180,E1 -1525.194,E2 -1525.194} C_VEL
LIN {X 0,Y 587.178,Z 1070.979,A -85,B 0,C 180,E1 -1526.569,E2 -1526.569} C_VEL
LIN {X 0,Y 587.127,Z 1072.89,A -85,B 0,C 180,E1 -1527.942,E2 -1527.942} C_VEL
LIN {X 0,Y 587.137,Z 1073.85,A -85,B 0,C 180,E1 -1529.314,E2 -1529.314} C_VEL
LIN {X 0,Y 587.137,Z 1073.85,A -85,B 0,C 180,E1 -1530.686,E2 -1530.686} C_VEL
LIN {X 0,Y 587.127,Z 1072.89,A -85,B 0,C 180,E1 -1532.058,E2 -1532.058} C_VEL
LIN {X 0,Y 587.178,Z 1070.979,A -85,B 0,C 180,E1 -1533.431,E2 -1533.431} C_VEL
LIN {X 0,Y 587.132,Z 1068.061,A -85,B 0,C 180,E1 -1534.806,E2 -1534.806} C_VEL
LIN {X 0,Y 587.16,Z 1064.115,A -85,B 0,C 180,E1 -1536.184,E2 -1536.184} C_VEL
LIN {X 0,Y 587.202,Z 1059.058,A -85,B 0,C 180,E1 -1537.565,E2 -1537.565} C_VEL
LIN {X 0,Y 587.248,Z 1052.858,A -85,B 0,C 180,E1 -1538.95,E2 -1538.95} C_VEL
LIN {X 0,Y 587.304,Z 1044.255,A -85,B 0,C 180,E1 -1540.515,E2 -1540.515} C_VEL
LIN {X 0,Y 587.364,Z 1034.97,A -85,B 0,C 180,E1 -1541.911,E2 -1541.911} C_VEL
LIN {X 0,Y 587.449,Z 1025.426,A -85,B 0,C 180,E1 -1543.138,E2 -1543.138} C_VEL
LIN {X 0,Y 587.591,Z 1013.571,A -85,B 0,C 180,E1 -1544.442,E2 -1544.442} C_VEL
LIN {X 0,Y 587.759,Z 1001.093,A -85,B 0,C 180,E1 -1545.607,E2 -1545.607} C_VEL
LIN {X 0,Y 587.904,Z 987.677,A -85,B 0,C 180,E1 -1546.672,E2 -1546.672} C_VEL
LIN {X 0,Y 588.063,Z 974.425,A -85,B 0,C 180,E1 -1547.563,E2 -1547.563} C_VEL
LIN {X 0,Y 588.237,Z 960.287,A -85,B 0,C 180,E1 -1548.367,E2 -1548.367} C_VEL
LIN {X 0,Y 588.451,Z 944.527,A -85,B 0,C 180,E1 -1549.104,E2 -1549.104} C_VEL
LIN {X 0,Y 588.623,Z 927.938,A -85,B 0,C 180,E1 -1549.712,E2 -1549.712} C_VEL
LIN {X 0,Y 588.707,Z 912.472,A -85,B 0,C 180,E1 -1550.141,E2 -1550.141} C_VEL
LIN {X 0,Y 588.786,Z 897.471,A -85,B 0,C 180,E1 -1550.434,E2 -1550.434} C_VEL
LIN {X 0,Y 589.25,Z 701.251,A -85,B 0,C 180,E1 -1552.953,E2 -1552.953} C_VEL
LIN {X 0,Y 588.093,Z 695.963,A -85,B 0,C 180,E1 -1553.087,E2 -1553.087} C_VEL
LIN {X 0,Y 588.196,Z 675.734,A -85,B 0,C 180,E1 -1555.666,E2 -1555.666} C_VEL
LIN {X 0,Y 588.468,Z 655.33,A -85,B 0,C 180,E1 -1558.341,E2 -1558.341} C_VEL
LIN {X 0,Y 588.396,Z 649.593,A -85,B 0,C 180,E1 -1559.112,E2 -1559.112} C_VEL
LIN {X 0,Y 587.354,Z 645.216,A -85,B 0,C 180,E1 -1559.797,E2 -1559.797} C_VEL
LIN {X 0,Y 587.338,Z 645.127,A -85,B 0,C 180,E1 -1562.578,E2 -1562.578} C_VEL
LIN {X 0,Y 587.345,Z 645.138,A -85,B 0,C 180,E1 -1565.053,E2 -1565.053} C_VEL
LIN {X 0,Y 587.335,Z 645.131,A -85,B 0,C 180,E1 -1567.838,E2 -1567.838} C_VEL
LIN {X 0,Y 587.314,Z 645.132,A -85,B 0,C 180,E1 -1570.253,E2 -1570.253} C_VEL
LIN {X 0,Y 587.319,Z 645.137,A -85,B 0,C 180,E1 -1573.119,E2 -1573.119} C_VEL
LIN {X 0,Y 587.328,Z 645.134,A -85,B 0,C 180,E1 -1576.05,E2 -1576.05} C_VEL
LIN {X 0,Y 587.357,Z 645.125,A -85,B 0,C 180,E1 -1578.921,E2 -1578.921} C_VEL
LIN {X 0,Y 587.33,Z 645.136,A -85,B 0,C 180,E1 -1581.521,E2 -1581.521} C_VEL
LIN {X 0,Y 587.345,Z 645.129,A -85,B 0,C 180,E1 -1584.454,E2 -1584.454} C_VEL
LIN {X 0,Y 587.332,Z 645.13,A -85,B 0,C 180,E1 -1586.887,E2 -1586.887} C_VEL
LIN {X 0,Y 587.342,Z 645.129,A -85,B 0,C 180,E1 -1589.487,E2 -1589.487} C_VEL
LIN {X 0,Y 587.342,Z 645.137,A -85,B 0,C 180,E1 -1592.306,E2 -1592.306} C_VEL
LIN {X 0,Y 587.335,Z 645.138,A -85,B 0,C 180,E1 -1594.483,E2 -1594.483} C_VEL
LIN {X 0,Y 587.337,Z 645.128,A -85,B 0,C 180,E1 -1597.486,E2 -1597.486} C_VEL
LIN {X 0,Y 587.325,Z 645.131,A -85,B 0,C 180,E1 -1599.695,E2 -1599.695} C_VEL
LIN {X 0,Y 587.352,Z 645.137,A -85,B 0,C 180,E1 -1602.594,E2 -1602.594} C_VEL
LIN {X 0,Y 587.354,Z 645.127,A -85,B 0,C 180,E1 -1605.738,E2 -1605.738} C_VEL
LIN {X 0,Y 587.35,Z 645.138,A -85,B 0,C 180,E1 -1608.858,E2 -1608.858} C_VEL
LIN {X 0,Y 587.363,Z 645.125,A -85,B 0,C 180,E1 -1611.745,E2 -1611.745} C_VEL
LIN {X 0,Y 587.358,Z 645.128,A -85,B 0,C 180,E1 -1614.507,E2 -1614.507} C_VEL
LIN {X 0,Y 587.375,Z 645.134,A -85,B 0,C 180,E1 -1617.257,E2 -1617.257} C_VEL
LIN {X 0,Y 587.371,Z 645.126,A -85,B 0,C 180,E1 -1620,E2 -1620} C_VEL
LIN {X 0,Y 587.374,Z 645.124,A -85,B 0,C 180,E1 -1622.743,E2 -1622.743} C_VEL
LIN {X 0,Y 587.358,Z 645.137,A -85,B 0,C 180,E1 -1625.493,E2 -1625.493} C_VEL
LIN {X 0,Y 587.363,Z 645.128,A -85,B 0,C 180,E1 -1628.255,E2 -1628.255} C_VEL
LIN {X 0,Y 587.35,Z 645.129,A -85,B 0,C 180,E1 -1631.141,E2 -1631.141} C_VEL
LIN {X 0,Y 587.354,Z 645.133,A -85,B 0,C 180,E1 -1634.261,E2 -1634.261} C_VEL
LIN {X 0,Y 587.351,Z 645.128,A -85,B 0,C 180,E1 -1637.406,E2 -1637.406} C_VEL
LIN {X 0,Y 587.318,Z 645.138,A -85,B 0,C 180,E1 -1638.32,E2 -1638.32} C_VEL
LIN {X 0,Y 586.661,Z 645.216,A -85,B 0,C 180,E1 -1638.892,E2 -1638.892} C_VEL
LIN {X 0,Y 583.826,Z 645.572,A -85,B 0,C 180,E1 -1639.82,E2 -1639.82} C_VEL
LIN {X 0,Y 581.418,Z 645.871,A -85,B 0,C 180,E1 -1640.567,E2 -1640.567} C_VEL
LIN {X 0,Y 580.371,Z 645.997,A -85,B 0,C 180,E1 -1641.144,E2 -1641.144} C_VEL
LIN {X 0,Y 580.28,Z 646.008,A -85,B 0,C 180,E1 -1641.339,E2 -1641.339} C_VEL
LIN {X 0,Y 580.292,Z 646.007,A -85,B 0,C 180,E1 -1643.557,E2 -1643.557} C_VEL
LIN {X 0,Y 580.318,Z 646.014,A -85,B 0,C 180,E1 -1646.342,E2 -1646.342} C_VEL
LIN {X 0,Y 580.299,Z 646.002,A -85,B 0,C 180,E1 -1649.312,E2 -1649.312} C_VEL
LIN {X 0,Y 580.293,Z 646.01,A -85,B 0,C 180,E1 -1652.2,E2 -1652.2} C_VEL
LIN {X 0,Y 580.293,Z 646.016,A -85,B 0,C 180,E1 -1654.696,E2 -1654.696} C_VEL
LIN {X 0,Y 580.292,Z 646.01,A -85,B 0,C 180,E1 -1657.268,E2 -1657.268} C_VEL
LIN {X 0,Y 580.299,Z 646.007,A -85,B 0,C 180,E1 -1660.273,E2 -1660.273} C_VEL
LIN {X 0,Y 580.289,Z 646.012,A -85,B 0,C 180,E1 -1662.705,E2 -1662.705} C_VEL
LIN {X 0,Y 580.264,Z 646.015,A -85,B 0,C 180,E1 -1665.609,E2 -1665.609} C_VEL
LIN {X 0,Y 580.305,Z 646.006,A -85,B 0,C 180,E1 -1668.235,E2 -1668.235} C_VEL
LIN {X 0,Y 580.281,Z 646.012,A -85,B 0,C 180,E1 -1670.967,E2 -1670.967} C_VEL
LIN {X 0,Y 580.289,Z 646.018,A -85,B 0,C 180,E1 -1673.599,E2 -1673.599} C_VEL
LIN {X 0,Y 580.312,Z 646.008,A -85,B 0,C 180,E1 -1676.146,E2 -1676.146} C_VEL
LIN {X 0,Y 580.285,Z 646.008,A -85,B 0,C 180,E1 -1678.616,E2 -1678.616} C_VEL
LIN {X 0,Y 580.287,Z 646.009,A -85,B 0,C 180,E1 -1681.024,E2 -1681.024} C_VEL
LIN {X 0,Y 580.286,Z 646.015,A -85,B 0,C 180,E1 -1683.666,E2 -1683.666} C_VEL
LIN {X 0,Y 580.297,Z 646.012,A -85,B 0,C 180,E1 -1685.684,E2 -1685.684} C_VEL
LIN {X 0,Y 580.268,Z 646.019,A -85,B 0,C 180,E1 -1687.948,E2 -1687.948} C_VEL
LIN {X 0,Y 580.314,Z 646.006,A -85,B 0,C 180,E1 -1690.914,E2 -1690.914} C_VEL
LIN {X 0,Y 580.275,Z 646.012,A -85,B 0,C 180,E1 -1693.826,E2 -1693.826} C_VEL
LIN {X 0,Y 580.321,Z 646.008,A -85,B 0,C 180,E1 -1695.983,E2 -1695.983} C_VEL
LIN {X 0,Y 580.3,Z 646.013,A -85,B 0,C 180,E1 -1698.827,E2 -1698.827} C_VEL
LIN {X 0,Y 580.329,Z 646.003,A -85,B 0,C 180,E1 -1701.644,E2 -1701.644} C_VEL
LIN {X 0,Y 580.323,Z 646.009,A -85,B 0,C 180,E1 -1704.44,E2 -1704.44} C_VEL
LIN {X 0,Y 580.334,Z 646.008,A -85,B 0,C 180,E1 -1707.224,E2 -1707.224} C_VEL
LIN {X 0,Y 580.351,Z 646.001,A -85,B 0,C 180,E1 -1710,E2 -1710} C_VEL
LIN {X 0,Y 580.334,Z 646.008,A -85,B 0,C 180,E1 -1712.776,E2 -1712.776} C_VEL
LIN {X 0,Y 580.323,Z 646.009,A -85,B 0,C 180,E1 -1715.56,E2 -1715.56} C_VEL
LIN {X 0,Y 580.329,Z 646.003,A -85,B 0,C 180,E1 -1718.356,E2 -1718.356} C_VEL
LIN {X 0,Y 580.296,Z 646.014,A -85,B 0,C 180,E1 -1721.191,E2 -1721.191} C_VEL
LIN {X 0,Y 580.321,Z 646.008,A -85,B 0,C 180,E1 -1724.017,E2 -1724.017} C_VEL
LIN {X 0,Y 580.307,Z 646.006,A -85,B 0,C 180,E1 -1726.913,E2 -1726.913} C_VEL
LIN {X 0,Y 580.3,Z 646.017,A -85,B 0,C 180,E1 -1729.822,E2 -1729.822} C_VEL
LIN {X 0,Y 580.29,Z 646.008,A -85,B 0,C 180,E1 -1732.802,E2 -1732.802} C_VEL
LIN {X 0,Y 580.301,Z 646.006,A -85,B 0,C 180,E1 -1735.079,E2 -1735.079} C_VEL
LIN {X 0,Y 580.295,Z 646.017,A -85,B 0,C 180,E1 -1738.185,E2 -1738.185} C_VEL
LIN {X 0,Y 580.294,Z 646.011,A -85,B 0,C 180,E1 -1740.697,E2 -1740.697} C_VEL
LIN {X 0,Y 580.298,Z 646.007,A -85,B 0,C 180,E1 -1743.316,E2 -1743.316} C_VEL
LIN {X 0,Y 580.318,Z 646.005,A -85,B 0,C 180,E1 -1745.767,E2 -1745.767} C_VEL
LIN {X 0,Y 580.28,Z 646.013,A -85,B 0,C 180,E1 -1748.146,E2 -1748.146} C_VEL
LIN {X 0,Y 580.293,Z 646.015,A -85,B 0,C 180,E1 -1750.843,E2 -1750.843} C_VEL
LIN {X 0,Y 580.278,Z 646.009,A -85,B 0,C 180,E1 -1753.656,E2 -1753.656} C_VEL
LIN {X 0,Y 580.283,Z 646.015,A -85,B 0,C 180,E1 -1756.607,E2 -1756.607} C_VEL
LIN {X 0,Y 580.311,Z 646.013,A -85,B 0,C 180,E1 -1759.158,E2 -1759.158} C_VEL
LIN {X 0,Y 580.282,Z 646.007,A -85,B 0,C 180,E1 -1761.926,E2 -1761.926} C_VEL
LIN {X 0,Y 580.299,Z 646.002,A -85,B 0,C 180,E1 -1764.457,E2 -1764.457} C_VEL
LIN {X 0,Y 580.282,Z 646.013,A -85,B 0,C 180,E1 -1766.975,E2 -1766.975} C_VEL
LIN {X 0,Y 580.299,Z 646.013,A -85,B 0,C 180,E1 -1769.426,E2 -1769.426} C_VEL
LIN {X 0,Y 580.309,Z 646.003,A -85,B 0,C 180,E1 -1772.136,E2 -1772.136} C_VEL
LIN {X 0,Y 580.299,Z 646.007,A -85,B 0,C 180,E1 -1774.92,E2 -1774.92} C_VEL
LIN {X 0,Y 580.318,Z 646.006,A -85,B 0,C 180,E1 -1777.199,E2 -1777.199} C_VEL
LIN {X 0,Y 580.299,Z 646.011,A -85,B 0,C 180,E1 -1780.178,E2 -1780.178} C_VEL
LIN {X 0,Y 580.318,Z 646.003,A -85,B 0,C 180,E1 -1783.103,E2 -1783.103} C_VEL
LIN {X 0,Y 580.317,Z 646.013,A -85,B 0,C 180,E1 -1785.983,E2 -1785.983} C_VEL
LIN {X 0,Y 580.319,Z 646.005,A -85,B 0,C 180,E1 -1788.827,E2 -1788.827} C_VEL
LIN {X 0,Y 580.326,Z 646.003,A -85,B 0,C 180,E1 -1791.644,E2 -1791.644} C_VEL
LIN {X 0,Y 580.324,Z 646.014,A -85,B 0,C 180,E1 -1794.44,E2 -1794.44} C_VEL
LIN {X 0,Y 580.339,Z 646,A -85,B 0,C 180,E1 -1797.224,E2 -1797.224} C_VEL
LIN {X 0,Y 580.34,Z 646.002,A -85,B 0,C 180,E1 -1800,E2 -1800} C_VEL
LIN {X 0,Y 580.34,Z 646.01,A -85,B 0,C 180,E1 -1802.777,E2 -1802.777} C_VEL
LIN {X 0,Y 580.325,Z 646.004,A -85,B 0,C 180,E1 -1805.56,E2 -1805.56} C_VEL
LIN {X 0,Y 580.326,Z 646.002,A -85,B 0,C 180,E1 -1808.356,E2 -1808.356} C_VEL
LIN {X 0,Y 580.322,Z 646.011,A -85,B 0,C 180,E1 -1811.209,E2 -1811.209} C_VEL
LIN {X 0,Y 580.318,Z 646.003,A -85,B 0,C 180,E1 -1814.017,E2 -1814.017} C_VEL
LIN {X 0,Y 580.302,Z 646.009,A -85,B 0,C 180,E1 -1816.915,E2 -1816.915} C_VEL
LIN {X 0,Y 580.299,Z 646.011,A -85,B 0,C 180,E1 -1819.823,E2 -1819.823} C_VEL
LIN {X 0,Y 580.268,Z 646.011,A -85,B 0,C 180,E1 -1822.053,E2 -1822.053} C_VEL
LIN {X 0,Y 580.301,Z 646.008,A -85,B 0,C 180,E1 -1825.08,E2 -1825.08} C_VEL
LIN {X 0,Y 580.311,Z 646.007,A -85,B 0,C 180,E1 -1827.864,E2 -1827.864} C_VEL
LIN {X 0,Y 580.29,Z 646.006,A -85,B 0,C 180,E1 -1830.698,E2 -1830.698} C_VEL
LIN {X 0,Y 580.297,Z 646.008,A -85,B 0,C 180,E1 -1833.318,E2 -1833.318} C_VEL
LIN {X 0,Y 580.32,Z 646.006,A -85,B 0,C 180,E1 -1835.768,E2 -1835.768} C_VEL
LIN {X 0,Y 580.284,Z 646.018,A -85,B 0,C 180,E1 -1838.147,E2 -1838.147} C_VEL
LIN {X 0,Y 580.313,Z 646.004,A -85,B 0,C 180,E1 -1840.842,E2 -1840.842} C_VEL
LIN {X 0,Y 580.284,Z 646.009,A -85,B 0,C 180,E1 -1843.657,E2 -1843.657} C_VEL
LIN {X 0,Y 580.279,Z 646.019,A -85,B 0,C 180,E1 -1846.609,E2 -1846.609} C_VEL
LIN {X 0,Y 580.295,Z 646.009,A -85,B 0,C 180,E1 -1849.158,E2 -1849.158} C_VEL
LIN {X 0,Y 580.285,Z 646.008,A -85,B 0,C 180,E1 -1851.928,E2 -1851.928} C_VEL
LIN {X 0,Y 580.301,Z 646.005,A -85,B 0,C 180,E1 -1854.457,E2 -1854.457} C_VEL
LIN {X 0,Y 580.288,Z 646.009,A -85,B 0,C 180,E1 -1856.976,E2 -1856.976} C_VEL
LIN {X 0,Y 580.351,Z 646.224,A -85,B 0,C 180,E1 -1859.957,E2 -1859.957} C_VEL
LIN {X 0,Y 581.731,Z 652.803,A -85,B 0,C 180,E1 -1860.958,E2 -1860.958} C_VEL
LIN {X 0,Y 581.474,Z 672.289,A -85,B 0,C 180,E1 -1863.56,E2 -1863.56} C_VEL
LIN {X 0,Y 581.231,Z 693.224,A -85,B 0,C 180,E1 -1866.295,E2 -1866.295} C_VEL
LIN {X 0,Y 581.219,Z 695.961,A -85,B 0,C 180,E1 -1866.623,E2 -1866.623} C_VEL
LIN {X 0,Y 582.694,Z 702.301,A -85,B 0,C 180,E1 -1866.788,E2 -1866.788} C_VEL
LIN {X 0,Y 582.149,Z 897.444,A -85,B 0,C 180,E1 -1869.322,E2 -1869.322} C_VEL
LIN {X 0,Y 582.041,Z 913.399,A -85,B 0,C 180,E1 -1869.641,E2 -1869.641} C_VEL
LIN {X 0,Y 581.895,Z 929.395,A -85,B 0,C 180,E1 -1870.097,E2 -1870.097} C_VEL
LIN {X 0,Y 581.696,Z 945.169,A -85,B 0,C 180,E1 -1870.692,E2 -1870.692} C_VEL
LIN {X 0,Y 581.465,Z 960.292,A -85,B 0,C 180,E1 -1871.411,E2 -1871.411} C_VEL
LIN {X 0,Y 581.226,Z 974.416,A -85,B 0,C 180,E1 -1872.223,E2 -1872.223} C_VEL
LIN {X 0,Y 581.032,Z 987.666,A -85,B 0,C 180,E1 -1873.125,E2 -1873.125} C_VEL
LIN {X 0,Y 580.824,Z 1001.093,A -85,B 0,C 180,E1 -1874.202,E2 -1874.202} C_VEL
LIN {X 0,Y 580.632,Z 1013.945,A -85,B 0,C 180,E1 -1875.418,E2 -1875.418} C_VEL
LIN {X 0,Y 580.441,Z 1025.427,A -85,B 0,C 180,E1 -1876.7,E2 -1876.7} C_VEL
LIN {X 0,Y 580.334,Z 1034.971,A -85,B 0,C 180,E1 -1877.942,E2 -1877.942} C_VEL
LIN {X 0,Y 580.232,Z 1044.254,A -85,B 0,C 180,E1 -1879.356,E2 -1879.356} C_VEL
LIN {X 0,Y 580.182,Z 1052.857,A -85,B 0,C 180,E1 -1880.94,E2 -1880.94} C_VEL
LIN {X 0,Y 580.118,Z 1059.061,A -85,B 0,C 180,E1 -1882.342,E2 -1882.342} C_VEL
LIN {X 0,Y 580.078,Z 1064.111,A -85,B 0,C 180,E1 -1883.74,E2 -1883.74} C_VEL
LIN {X 0,Y 580.035,Z 1068.062,A -85,B 0,C 180,E1 -1885.135,E2 -1885.135} C_VEL
LIN {X 0,Y 580.104,Z 1070.975,A -85,B 0,C 180,E1 -1886.527,E2 -1886.527} C_VEL
LIN {X 0,Y 580.026,Z 1072.891,A -85,B 0,C 180,E1 -1887.917,E2 -1887.917} C_VEL
LIN {X 0,Y 580.037,Z 1073.848,A -85,B 0,C 180,E1 -1889.306,E2 -1889.306} C_VEL
LIN {X 0,Y 580.037,Z 1073.848,A -85,B 0,C 180,E1 -1890.694,E2 -1890.694} C_VEL
LIN {X 0,Y 580.026,Z 1072.891,A -85,B 0,C 180,E1 -1892.083,E2 -1892.083} C_VEL
LIN {X 0,Y 580.104,Z 1070.975,A -85,B 0,C 180,E1 -1893.473,E2 -1893.473} C_VEL
LIN {X 0,Y 580.035,Z 1068.062,A -85,B 0,C 180,E1 -1894.865,E2 -1894.865} C_VEL
LIN {X 0,Y 580.075,Z 1064.111,A -85,B 0,C 180,E1 -1896.26,E2 -1896.26} C_VEL
LIN {X 0,Y 580.118,Z 1059.061,A -85,B 0,C 180,E1 -1897.658,E2 -1897.658} C_VEL
LIN {X 0,Y 580.182,Z 1052.857,A -85,B 0,C 180,E1 -1899.06,E2 -1899.06} C_VEL
LIN {X 0,Y 580.232,Z 1044.254,A -85,B 0,C 180,E1 -1900.644,E2 -1900.644} C_VEL
LIN {X 0,Y 580.334,Z 1034.971,A -85,B 0,C 180,E1 -1902.058,E2 -1902.058} C_VEL
LIN {X 0,Y 580.441,Z 1025.427,A -85,B 0,C 180,E1 -1903.3,E2 -1903.3} C_VEL
LIN {X 0,Y 580.632,Z 1013.947,A -85,B 0,C 180,E1 -1904.582,E2 -1904.582} C_VEL
LIN {X 0,Y 580.824,Z 1001.093,A -85,B 0,C 180,E1 -1905.798,E2 -1905.798} C_VEL
LIN {X 0,Y 581.023,Z 987.666,A -85,B 0,C 180,E1 -1906.876,E2 -1906.876} C_VEL
LIN {X 0,Y 581.226,Z 974.416,A -85,B 0,C 180,E1 -1907.777,E2 -1907.777} C_VEL
LIN {X 0,Y 581.464,Z 960.292,A -85,B 0,C 180,E1 -1908.589,E2 -1908.589} C_VEL
LIN {X 0,Y 581.706,Z 945.116,A -85,B 0,C 180,E1 -1909.31,E2 -1909.31} C_VEL
LIN {X 0,Y 581.885,Z 927.922,A -85,B 0,C 180,E1 -1909.95,E2 -1909.95} C_VEL
LIN {X 0,Y 582.053,Z 912.443,A -85,B 0,C 180,E1 -1910.381,E2 -1910.381} C_VEL
LIN {X 0,Y 582.159,Z 897.444,A -85,B 0,C 180,E1 -1910.677,E2 -1910.677} C_VEL
LIN {X 0,Y 582.719,Z 703.595,A -85,B 0,C 180,E1 -1913.194,E2 -1913.194} C_VEL
LIN {X 0,Y 581.964,Z 699.141,A -85,B 0,C 180,E1 -1913.285,E2 -1913.285} C_VEL
LIN {X 0,Y 581.204,Z 695.845,A -85,B 0,C 180,E1 -1913.385,E2 -1913.385} C_VEL
LIN {X 0,Y 581.393,Z 677.192,A -85,B 0,C 180,E1 -1915.796,E2 -1915.796} C_VEL
LIN {X 0,Y 581.71,Z 656.786,A -85,B 0,C 180,E1 -1918.503,E2 -1918.503} C_VEL
LIN {X 0,Y 581.681,Z 651.732,A -85,B 0,C 180,E1 -1919.19,E2 -1919.19} C_VEL
LIN {X 0,Y 580.322,Z 646.099,A -85,B 0,C 180,E1 -1920.07,E2 -1920.07} C_VEL
LIN {X 0,Y 580.288,Z 646.009,A -85,B 0,C 180,E1 -1923.024,E2 -1923.024} C_VEL
LIN {X 0,Y 580.321,Z 646,A -85,B 0,C 180,E1 -1925.767,E2 -1925.767} C_VEL
LIN {X 0,Y 580.283,Z 646.008,A -85,B 0,C 180,E1 -1928.146,E2 -1928.146} C_VEL
LIN {X 0,Y 580.295,Z 646.009,A -85,B 0,C 180,E1 -1930.842,E2 -1930.842} C_VEL
LIN {X 0,Y 580.281,Z 646.014,A -85,B 0,C 180,E1 -1933.656,E2 -1933.656} C_VEL
LIN {X 0,Y 580.286,Z 646.008,A -85,B 0,C 180,E1 -1936.607,E2 -1936.607} C_VEL
LIN {X 0,Y 580.313,Z 646.004,A -85,B 0,C 180,E1 -1939.158,E2 -1939.158} C_VEL
LIN {X 0,Y 580.285,Z 646.016,A -85,B 0,C 180,E1 -1941.926,E2 -1941.926} C_VEL
LIN {X 0,Y 580.3,Z 646.006,A -85,B 0,C 180,E1 -1944.456,E2 -1944.456} C_VEL
LIN {X 0,Y 580.284,Z 646.008,A -85,B 0,C 180,E1 -1946.975,E2 -1946.975} C_VEL
LIN {X 0,Y 580.301,Z 646.006,A -85,B 0,C 180,E1 -1949.425,E2 -1949.425} C_VEL
LIN {X 0,Y 580.311,Z 646.007,A -85,B 0,C 180,E1 -1952.136,E2 -1952.136} C_VEL
LIN {X 0,Y 580.301,Z 646.008,A -85,B 0,C 180,E1 -1954.92,E2 -1954.92} C_VEL
LIN {X 0,Y 580.268,Z 646.011,A -85,B 0,C 180,E1 -1957.947,E2 -1957.947} C_VEL
LIN {X 0,Y 580.307,Z 646.009,A -85,B 0,C 180,E1 -1960.914,E2 -1960.914} C_VEL
LIN {X 0,Y 580.279,Z 646.008,A -85,B 0,C 180,E1 -1963.826,E2 -1963.826} C_VEL
LIN {X 0,Y 580.273,Z 646.018,A -85,B 0,C 180,E1 -1966.696,E2 -1966.696} C_VEL
LIN {X 0,Y 580.298,Z 646.008,A -85,B 0,C 180,E1 -1969.533,E2 -1969.533} C_VEL
LIN {X 0,Y 580.331,Z 646.001,A -85,B 0,C 180,E1 -1972.345,E2 -1972.345} C_VEL
LIN {X 0,Y 580.334,Z 646.013,A -85,B 0,C 180,E1 -1975.137,E2 -1975.137} C_VEL
LIN {X 0,Y 580.329,Z 646.003,A -85,B 0,C 180,E1 -1977.918,E2 -1977.918} C_VEL
LIN {X 0,Y 580.359,Z 646,A -85,B 0,C 180,E1 -1980.694,E2 -1980.694} C_VEL
LIN {X 0,Y 580.282,Z 646.017,A -85,B 0,C 180,E1 -1983.472,E2 -1983.472} C_VEL
LIN {X 0,Y 580.324,Z 646.014,A -85,B 0,C 180,E1 -1985.56,E2 -1985.56} C_VEL
LIN {X 0,Y 580.326,Z 646.003,A -85,B 0,C 180,E1 -1988.356,E2 -1988.356} C_VEL
LIN {X 0,Y 580.321,Z 646.005,A -85,B 0,C 180,E1 -1991.208,E2 -1991.208} C_VEL
LIN {X 0,Y 580.304,Z 646.01,A -85,B 0,C 180,E1 -1994.339,E2 -1994.339} C_VEL
LIN {X 0,Y 580.302,Z 646.005,A -85,B 0,C 180,E1 -1996.915,E2 -1996.915} C_VEL
LIN {X 0,Y 580.299,Z 646.011,A -85,B 0,C 180,E1 -1999.822,E2 -1999.822} C_VEL
LIN {X 0,Y 580.28,Z 646.008,A -85,B 0,C 180,E1 -2001.339,E2 -2001.339} C_VEL
LIN {X 0,Y 579.59,Z 646.101,A -85,B 0,C 180,E1 -2001.918,E2 -2001.918} C_VEL
LIN {X 0,Y 576.717,Z 646.454,A -85,B 0,C 180,E1 -2002.858,E2 -2002.858} C_VEL
LIN {X 0,Y 574.318,Z 646.752,A -85,B 0,C 180,E1 -2003.615,E2 -2003.615} C_VEL
LIN {X 0,Y 573.313,Z 646.885,A -85,B 0,C 180,E1 -2004.199,E2 -2004.199} C_VEL
LIN {X 0,Y 573.244,Z 646.889,A -85,B 0,C 180,E1 -2004.397,E2 -2004.397} C_VEL
LIN {X 0,Y 573.254,Z 646.882,A -85,B 0,C 180,E1 -2006.975,E2 -2006.975} C_VEL
LIN {X 0,Y 573.245,Z 646.88,A -85,B 0,C 180,E1 -2009.49,E2 -2009.49} C_VEL
LIN {X 0,Y 573.246,Z 646.888,A -85,B 0,C 180,E1 -2012.23,E2 -2012.23} C_VEL
LIN {X 0,Y 573.244,Z 646.891,A -85,B 0,C 180,E1 -2014.775,E2 -2014.775} C_VEL
LIN {X 0,Y 573.245,Z 646.889,A -85,B 0,C 180,E1 -2017.167,E2 -2017.167} C_VEL
LIN {X 0,Y 573.242,Z 646.887,A -85,B 0,C 180,E1 -2019.607,E2 -2019.607} C_VEL
LIN {X 0,Y 573.251,Z 646.888,A -85,B 0,C 180,E1 -2022.644,E2 -2022.644} C_VEL
LIN {X 0,Y 573.23,Z 646.891,A -85,B 0,C 180,E1 -2025.667,E2 -2025.667} C_VEL
LIN {X 0,Y 573.236,Z 646.887,A -85,B 0,C 180,E1 -2028.545,E2 -2028.545} C_VEL
LIN {X 0,Y 573.24,Z 646.895,A -85,B 0,C 180,E1 -2031.299,E2 -2031.299} C_VEL
LIN {X 0,Y 573.256,Z 646.887,A -85,B 0,C 180,E1 -2034.012,E2 -2034.012} C_VEL
LIN {X 0,Y 573.278,Z 646.882,A -85,B 0,C 180,E1 -2036.519,E2 -2036.519} C_VEL
LIN {X 0,Y 573.238,Z 646.888,A -85,B 0,C 180,E1 -2039.115,E2 -2039.115} C_VEL
LIN {X 0,Y 573.257,Z 646.893,A -85,B 0,C 180,E1 -2041.969,E2 -2041.969} C_VEL
LIN {X 0,Y 573.249,Z 646.887,A -85,B 0,C 180,E1 -2044.59,E2 -2044.59} C_VEL
LIN {X 0,Y 573.232,Z 646.891,A -85,B 0,C 180,E1 -2047.663,E2 -2047.663} C_VEL
LIN {X 0,Y 573.273,Z 646.885,A -85,B 0,C 180,E1 -2050.729,E2 -2050.729} C_VEL
LIN {X 0,Y 573.247,Z 646.886,A -85,B 0,C 180,E1 -2053.622,E2 -2053.622} C_VEL
LIN {X 0,Y 573.268,Z 646.885,A -85,B 0,C 180,E1 -2055.807,E2 -2055.807} C_VEL
LIN {X 0,Y 573.258,Z 646.892,A -85,B 0,C 180,E1 -2058.745,E2 -2058.745} C_VEL
LIN {X 0,Y 573.285,Z 646.881,A -85,B 0,C 180,E1 -2061.541,E2 -2061.541} C_VEL
LIN {X 0,Y 573.289,Z 646.884,A -85,B 0,C 180,E1 -2064.372,E2 -2064.372} C_VEL
LIN {X 0,Y 573.308,Z 646.878,A -85,B 0,C 180,E1 -2067.892,E2 -2067.892} C_VEL
LIN {X 0,Y 573.327,Z 646.881,A -85,B 0,C 180,E1 -2070.702,E2 -2070.702} C_VEL
LIN {X 0,Y 573.237,Z 646.892,A -85,B 0,C 180,E1 -2073.514,E2 -2073.514} C_VEL
LIN {X 0,Y 573.289,Z 646.884,A -85,B 0,C 180,E1 -2075.628,E2 -2075.628} C_VEL
LIN {X 0,Y 573.285,Z 646.881,A -85,B 0,C 180,E1 -2078.459,E2 -2078.459} C_VEL
LIN {X 0,Y 573.267,Z 646.892,A -85,B 0,C 180,E1 -2081.312,E2 -2081.312} C_VEL
LIN {X 0,Y 573.277,Z 646.882,A -85,B 0,C 180,E1 -2084.424,E2 -2084.424} C_VEL
LIN {X 0,Y 573.254,Z 646.886,A -85,B 0,C 180,E1 -2087.111,E2 -2087.111} C_VEL
LIN {X 0,Y 573.248,Z 646.892,A -85,B 0,C 180,E1 -2090.076,E2 -2090.076} C_VEL
LIN {X 0,Y 573.228,Z 646.888,A -85,B 0,C 180,E1 -2093.099,E2 -2093.099} C_VEL
LIN {X 0,Y 573.249,Z 646.887,A -85,B 0,C 180,E1 -2095.41,E2 -2095.41} C_VEL
LIN {X 0,Y 573.258,Z 646.893,A -85,B 0,C 180,E1 -2098.031,E2 -2098.031} C_VEL
LIN {X 0,Y 573.238,Z 646.888,A -85,B 0,C 180,E1 -2100.885,E2 -2100.885} C_VEL
LIN {X 0,Y 573.254,Z 646.885,A -85,B 0,C 180,E1 -2103.524,E2 -2103.524} C_VEL
LIN {X 0,Y 573.253,Z 646.888,A -85,B 0,C 180,E1 -2106.048,E2 -2106.048} C_VEL
LIN {X 0,Y 573.24,Z 646.895,A -85,B 0,C 180,E1 -2108.701,E2 -2108.701} C_VEL
LIN {X 0,Y 573.245,Z 646.885,A -85,B 0,C 180,E1 -2111.595,E2 -2111.595} C_VEL
LIN {X 0,Y 573.23,Z 646.891,A -85,B 0,C 180,E1 -2114.333,E2 -2114.333} C_VEL
LIN {X 0,Y 573.251,Z 646.888,A -85,B 0,C 180,E1 -2117.356,E2 -2117.356} C_VEL
LIN {X 0,Y 573.242,Z 646.887,A -85,B 0,C 180,E1 -2120.393,E2 -2120.393} C_VEL
LIN {X 0,Y 573.247,Z 646.89,A -85,B 0,C 180,E1 -2123.078,E2 -2123.078} C_VEL
LIN {X 0,Y 573.266,Z 646.886,A -85,B 0,C 180,E1 -2125.672,E2 -2125.672} C_VEL
LIN {X 0,Y 573.24,Z 646.886,A -85,B 0,C 180,E1 -2128.185,E2 -2128.185} C_VEL
LIN {X 0,Y 573.261,Z 646.878,A -85,B 0,C 180,E1 -2130.634,E2 -2130.634} C_VEL
LIN {X 0,Y 573.26,Z 646.889,A -85,B 0,C 180,E1 -2133.5,E2 -2133.5} C_VEL
LIN {X 0,Y 573.234,Z 646.889,A -85,B 0,C 180,E1 -2136.135,E2 -2136.135} C_VEL
LIN {X 0,Y 573.249,Z 646.884,A -85,B 0,C 180,E1 -2138.706,E2 -2138.706} C_VEL
LIN {X 0,Y 573.229,Z 646.89,A -85,B 0,C 180,E1 -2141.412,E2 -2141.412} C_VEL
LIN {X 0,Y 573.25,Z 646.887,A -85,B 0,C 180,E1 -2143.622,E2 -2143.622} C_VEL
LIN {X 0,Y 573.228,Z 646.888,A -85,B 0,C 180,E1 -2146.53,E2 -2146.53} C_VEL
LIN {X 0,Y 573.271,Z 646.884,A -85,B 0,C 180,E1 -2148.734,E2 -2148.734} C_VEL
LIN {X 0,Y 573.297,Z 646.878,A -85,B 0,C 180,E1 -2151.541,E2 -2151.541} C_VEL
LIN {X 0,Y 573.292,Z 646.889,A -85,B 0,C 180,E1 -2154.372,E2 -2154.372} C_VEL
LIN {X 0,Y 573.299,Z 646.877,A -85,B 0,C 180,E1 -2157.893,E2 -2157.893} C_VEL
LIN {X 0,Y 573.331,Z 646.884,A -85,B 0,C 180,E1 -2160.703,E2 -2160.703} C_VEL
LIN {X 0,Y 573.233,Z 646.886,A -85,B 0,C 180,E1 -2163.515,E2 -2163.515} C_VEL
LIN {X 0,Y 573.292,Z 646.88,A -85,B 0,C 180,E1 -2165.628,E2 -2165.628} C_VEL
LIN {X 0,Y 573.298,Z 646.878,A -85,B 0,C 180,E1 -2168.459,E2 -2168.459} C_VEL
LIN {X 0,Y 573.288,Z 646.885,A -85,B 0,C 180,E1 -2171.312,E2 -2171.312} C_VEL
LIN {X 0,Y 573.27,Z 646.881,A -85,B 0,C 180,E1 -2174.425,E2 -2174.425} C_VEL
LIN {X 0,Y 573.249,Z 646.891,A -85,B 0,C 180,E1 -2177.112,E2 -2177.112} C_VEL
LIN {X 0,Y 573.248,Z 646.886,A -85,B 0,C 180,E1 -2180.077,E2 -2180.077} C_VEL
LIN {X 0,Y 573.232,Z 646.885,A -85,B 0,C 180,E1 -2182.338,E2 -2182.338} C_VEL
LIN {X 0,Y 573.25,Z 646.891,A -85,B 0,C 180,E1 -2185.41,E2 -2185.41} C_VEL
LIN {X 0,Y 573.255,Z 646.882,A -85,B 0,C 180,E1 -2188.032,E2 -2188.032} C_VEL
LIN {X 0,Y 573.235,Z 646.885,A -85,B 0,C 180,E1 -2190.886,E2 -2190.886} C_VEL
LIN {X 0,Y 573.279,Z 646.884,A -85,B 0,C 180,E1 -2193.529,E2 -2193.529} C_VEL
LIN {X 0,Y 573.254,Z 646.889,A -85,B 0,C 180,E1 -2196.049,E2 -2196.049} C_VEL
LIN {X 0,Y 573.244,Z 646.888,A -85,B 0,C 180,E1 -2198.701,E2 -2198.701} C_VEL
LIN {X 0,Y 573.258,Z 646.881,A -85,B 0,C 180,E1 -2201.598,E2 -2201.598} C_VEL
LIN {X 0,Y 573.232,Z 646.897,A -85,B 0,C 180,E1 -2204.334,E2 -2204.334} C_VEL
LIN {X 0,Y 573.237,Z 646.887,A -85,B 0,C 180,E1 -2207.359,E2 -2207.359} C_VEL
LIN {X 0,Y 573.242,Z 646.891,A -85,B 0,C 180,E1 -2210.394,E2 -2210.394} C_VEL
LIN {X 0,Y 573.252,Z 646.881,A -85,B 0,C 180,E1 -2213.079,E2 -2213.079} C_VEL
LIN {X 0,Y 573.269,Z 646.885,A -85,B 0,C 180,E1 -2215.672,E2 -2215.672} C_VEL
LIN {X 0,Y 573.247,Z 646.88,A -85,B 0,C 180,E1 -2218.186,E2 -2218.186} C_VEL
LIN {X 0,Y 573.31,Z 647.122,A -85,B 0,C 180,E1 -2219.676,E2 -2219.676} C_VEL
LIN {X 0,Y 574.949,Z 653.871,A -85,B 0,C 180,E1 -2220.729,E2 -2220.729} C_VEL
LIN {X 0,Y 574.707,Z 671.361,A -85,B 0,C 180,E1 -2223.099,E2 -2223.099} C_VEL
LIN {X 0,Y 574.386,Z 691.767,A -85,B 0,C 180,E1 -2225.802,E2 -2225.802} C_VEL
LIN {X 0,Y 574.37,Z 696.062,A -85,B 0,C 180,E1 -2226.333,E2 -2226.333} C_VEL
LIN {X 0,Y 576.203,Z 703.827,A -85,B 0,C 180,E1 -2226.531,E2 -2226.531} C_VEL
LIN {X 0,Y 575.5,Z 898.809,A -85,B 0,C 180,E1 -2229.096,E2 -2229.096} C_VEL
LIN {X 0,Y 575.378,Z 914.318,A -85,B 0,C 180,E1 -2229.418,E2 -2229.418} C_VEL
LIN {X 0,Y 575.155,Z 930.717,A -85,B 0,C 180,E1 -2229.9,E2 -2229.9} C_VEL
LIN {X 0,Y 574.919,Z 947.267,A -85,B 0,C 180,E1 -2230.551,E2 -2230.551} C_VEL
LIN {X 0,Y 574.651,Z 961.987,A -85,B 0,C 180,E1 -2231.275,E2 -2231.275} C_VEL
LIN {X 0,Y 574.382,Z 975.832,A -85,B 0,C 180,E1 -2232.096,E2 -2232.096} C_VEL
LIN {X 0,Y 574.127,Z 990.08,A -85,B 0,C 180,E1 -2233.099,E2 -2233.099} C_VEL
LIN {X 0,Y 573.88,Z 1003.134,A -85,B 0,C 180,E1 -2234.188,E2 -2234.188} C_VEL
LIN {X 0,Y 573.62,Z 1015.888,A -85,B 0,C 180,E1 -2235.445,E2 -2235.445} C_VEL
LIN {X 0,Y 573.419,Z 1026.883,A -85,B 0,C 180,E1 -2236.715,E2 -2236.715} C_VEL
LIN {X 0,Y 573.303,Z 1036.21,A -85,B 0,C 180,E1 -2237.972,E2 -2237.972} C_VEL
LIN {X 0,Y 573.163,Z 1045.277,A -85,B 0,C 180,E1 -2239.402,E2 -2239.402} C_VEL
LIN {X 0,Y 573.094,Z 1052.856,A -85,B 0,C 180,E1 -2240.827,E2 -2240.827} C_VEL
LIN {X 0,Y 573.056,Z 1059.063,A -85,B 0,C 180,E1 -2242.247,E2 -2242.247} C_VEL
LIN {X 0,Y 573.004,Z 1064.107,A -85,B 0,C 180,E1 -2243.663,E2 -2243.663} C_VEL
LIN {X 0,Y 572.944,Z 1068.064,A -85,B 0,C 180,E1 -2245.074,E2 -2245.074} C_VEL
LIN {X 0,Y 573.003,Z 1070.97,A -85,B 0,C 180,E1 -2246.484,E2 -2246.484} C_VEL
LIN {X 0,Y 572.926,Z 1072.891,A -85,B 0,C 180,E1 -2247.891,E2 -2247.891} C_VEL
LIN {X 0,Y 572.938,Z 1073.843,A -85,B 0,C 180,E1 -2249.297,E2 -2249.297} C_VEL
LIN {X 0,Y 572.938,Z 1073.843,A -85,B 0,C 180,E1 -2250.703,E2 -2250.703} C_VEL
LIN {X 0,Y 572.926,Z 1072.891,A -85,B 0,C 180,E1 -2252.109,E2 -2252.109} C_VEL
LIN {X 0,Y 573.003,Z 1070.97,A -85,B 0,C 180,E1 -2253.516,E2 -2253.516} C_VEL
LIN {X 0,Y 572.944,Z 1068.064,A -85,B 0,C 180,E1 -2254.926,E2 -2254.926} C_VEL
LIN {X 0,Y 573.004,Z 1064.107,A -85,B 0,C 180,E1 -2256.337,E2 -2256.337} C_VEL
LIN {X 0,Y 573.056,Z 1059.063,A -85,B 0,C 180,E1 -2257.753,E2 -2257.753} C_VEL
LIN {X 0,Y 573.094,Z 1052.856,A -85,B 0,C 180,E1 -2259.173,E2 -2259.173} C_VEL
LIN {X 0,Y 573.163,Z 1045.277,A -85,B 0,C 180,E1 -2260.598,E2 -2260.598} C_VEL
LIN {X 0,Y 573.303,Z 1036.21,A -85,B 0,C 180,E1 -2262.028,E2 -2262.028} C_VEL
LIN {X 0,Y 573.419,Z 1026.883,A -85,B 0,C 180,E1 -2263.285,E2 -2263.285} C_VEL
LIN {X 0,Y 573.617,Z 1015.898,A -85,B 0,C 180,E1 -2264.554,E2 -2264.554} C_VEL
LIN {X 0,Y 573.859,Z 1003.134,A -85,B 0,C 180,E1 -2265.812,E2 -2265.812} C_VEL
LIN {X 0,Y 574.13,Z 988.897,A -85,B 0,C 180,E1 -2266.993,E2 -2266.993} C_VEL
LIN {X 0,Y 574.382,Z 975.832,A -85,B 0,C 180,E1 -2267.904,E2 -2267.904} C_VEL
LIN {X 0,Y 574.651,Z 961.987,A -85,B 0,C 180,E1 -2268.725,E2 -2268.725} C_VEL
LIN {X 0,Y 574.922,Z 947.243,A -85,B 0,C 180,E1 -2269.45,E2 -2269.45} C_VEL
LIN {X 0,Y 575.16,Z 930.717,A -85,B 0,C 180,E1 -2270.1,E2 -2270.1} C_VEL
LIN {X 0,Y 575.377,Z 914.318,A -85,B 0,C 180,E1 -2270.582,E2 -2270.582} C_VEL
LIN {X 0,Y 575.498,Z 898.809,A -85,B 0,C 180,E1 -2270.904,E2 -2270.904} C_VEL
LIN {X 0,Y 576.187,Z 704.218,A -85,B 0,C 180,E1 -2273.464,E2 -2273.464} C_VEL
LIN {X 0,Y 574.4,Z 696.124,A -85,B 0,C 180,E1 -2273.662,E2 -2273.662} C_VEL
LIN {X 0,Y 574.508,Z 685.564,A -85,B 0,C 180,E1 -2275.012,E2 -2275.012} C_VEL
LIN {X 0,Y 574.884,Z 663.127,A -85,B 0,C 180,E1 -2278.007,E2 -2278.007} C_VEL
LIN {X 0,Y 574.948,Z 653.871,A -85,B 0,C 180,E1 -2279.271,E2 -2279.271} C_VEL
LIN {X 0,Y 573.288,Z 646.99,A -85,B 0,C 180,E1 -2280.351,E2 -2280.351} C_VEL
LIN {X 0,Y 573.281,Z 646.887,A -85,B 0,C 180,E1 -2283.48,E2 -2283.48} C_VEL
LIN {X 0,Y 573.256,Z 646.878,A -85,B 0,C 180,E1 -2286.047,E2 -2286.047} C_VEL
LIN {X 0,Y 573.243,Z 646.887,A -85,B 0,C 180,E1 -2288.7,E2 -2288.7} C_VEL
LIN {X 0,Y 573.248,Z 646.893,A -85,B 0,C 180,E1 -2291.595,E2 -2291.595} C_VEL
LIN {X 0,Y 573.232,Z 646.884,A -85,B 0,C 180,E1 -2294.332,E2 -2294.332} C_VEL
LIN {X 0,Y 573.254,Z 646.891,A -85,B 0,C 180,E1 -2297.355,E2 -2297.355} C_VEL
LIN {X 0,Y 573.244,Z 646.887,A -85,B 0,C 180,E1 -2300.393,E2 -2300.393} C_VEL
LIN {X 0,Y 573.249,Z 646.884,A -85,B 0,C 180,E1 -2303.077,E2 -2303.077} C_VEL
LIN {X 0,Y 573.268,Z 646.885,A -85,B 0,C 180,E1 -2305.671,E2 -2305.671} C_VEL
LIN {X 0,Y 573.242,Z 646.893,A -85,B 0,C 180,E1 -2308.185,E2 -2308.185} C_VEL
LIN {X 0,Y 573.263,Z 646.877,A -85,B 0,C 180,E1 -2310.634,E2 -2310.634} C_VEL
LIN {X 0,Y 573.262,Z 646.881,A -85,B 0,C 180,E1 -2313.5,E2 -2313.5} C_VEL
LIN {X 0,Y 573.224,Z 646.894,A -85,B 0,C 180,E1 -2316.134,E2 -2316.134} C_VEL
LIN {X 0,Y 573.252,Z 646.886,A -85,B 0,C 180,E1 -2319.174,E2 -2319.174} C_VEL
LIN {X 0,Y 573.229,Z 646.886,A -85,B 0,C 180,E1 -2321.411,E2 -2321.411} C_VEL
LIN {X 0,Y 573.253,Z 646.884,A -85,B 0,C 180,E1 -2323.622,E2 -2323.622} C_VEL
LIN {X 0,Y 573.231,Z 646.892,A -85,B 0,C 180,E1 -2326.529,E2 -2326.529} C_VEL
LIN {X 0,Y 573.267,Z 646.885,A -85,B 0,C 180,E1 -2329.403,E2 -2329.403} C_VEL
LIN {X 0,Y 573.28,Z 646.878,A -85,B 0,C 180,E1 -2332.25,E2 -2332.25} C_VEL
LIN {X 0,Y 573.306,Z 646.887,A -85,B 0,C 180,E1 -2335.077,E2 -2335.077} C_VEL
LIN {X 0,Y 573.3,Z 646.879,A -85,B 0,C 180,E1 -2337.892,E2 -2337.892} C_VEL
LIN {X 0,Y 573.329,Z 646.875,A -85,B 0,C 180,E1 -2340.702,E2 -2340.702} C_VEL
LIN {X 0,Y 573.234,Z 646.895,A -85,B 0,C 180,E1 -2343.514,E2 -2343.514} C_VEL
LIN {X 0,Y 573.292,Z 646.889,A -85,B 0,C 180,E1 -2345.628,E2 -2345.628} C_VEL
LIN {X 0,Y 573.297,Z 646.878,A -85,B 0,C 180,E1 -2348.459,E2 -2348.459} C_VEL
LIN {X 0,Y 573.287,Z 646.882,A -85,B 0,C 180,E1 -2351.311,E2 -2351.311} C_VEL
LIN {X 0,Y 573.27,Z 646.885,A -85,B 0,C 180,E1 -2354.425,E2 -2354.425} C_VEL
LIN {X 0,Y 573.248,Z 646.883,A -85,B 0,C 180,E1 -2357.112,E2 -2357.112} C_VEL
LIN {X 0,Y 573.247,Z 646.894,A -85,B 0,C 180,E1 -2360.076,E2 -2360.076} C_VEL
LIN {X 0,Y 573.26,Z 646.883,A -85,B 0,C 180,E1 -2363.154,E2 -2363.154} C_VEL
LIN {X 0,Y 573.244,Z 646.889,A -85,B 0,C 180,E1 -2364.397,E2 -2364.397} C_VEL
LIN {X 0,Y 572.612,Z 646.97,A -85,B 0,C 180,E1 -2364.983,E2 -2364.983} C_VEL
LIN {X 0,Y 569.772,Z 647.321,A -85,B 0,C 180,E1 -2365.935,E2 -2365.935} C_VEL
LIN {X 0,Y 567.346,Z 647.621,A -85,B 0,C 180,E1 -2366.701,E2 -2366.701} C_VEL
LIN {X 0,Y 566.295,Z 647.746,A -85,B 0,C 180,E1 -2367.292,E2 -2367.292} C_VEL
LIN {X 0,Y 566.206,Z 647.757,A -85,B 0,C 180,E1 -2367.492,E2 -2367.492} C_VEL
LIN {X 0,Y 566.217,Z 647.755,A -85,B 0,C 180,E1 -2369.767,E2 -2369.767} C_VEL
LIN {X 0,Y 566.198,Z 647.769,A -85,B 0,C 180,E1 -2372.431,E2 -2372.431} C_VEL
LIN {X 0,Y 566.205,Z 647.762,A -85,B 0,C 180,E1 -2374.995,E2 -2374.995} C_VEL
LIN {X 0,Y 566.187,Z 647.765,A -85,B 0,C 180,E1 -2377.461,E2 -2377.461} C_VEL
LIN {X 0,Y 566.218,Z 647.761,A -85,B 0,C 180,E1 -2380.198,E2 -2380.198} C_VEL
LIN {X 0,Y 566.203,Z 647.773,A -85,B 0,C 180,E1 -2383.053,E2 -2383.053} C_VEL
LIN {X 0,Y 566.193,Z 647.764,A -85,B 0,C 180,E1 -2386.049,E2 -2386.049} C_VEL
LIN {X 0,Y 566.203,Z 647.766,A -85,B 0,C 180,E1 -2388.864,E2 -2388.864} C_VEL
LIN {X 0,Y 566.181,Z 647.773,A -85,B 0,C 180,E1 -2391.638,E2 -2391.638} C_VEL
LIN {X 0,Y 566.204,Z 647.763,A -85,B 0,C 180,E1 -2394.312,E2 -2394.312} C_VEL
LIN {X 0,Y 566.222,Z 647.761,A -85,B 0,C 180,E1 -2396.899,E2 -2396.899} C_VEL
LIN {X 0,Y 566.188,Z 647.77,A -85,B 0,C 180,E1 -2399.409,E2 -2399.409} C_VEL
LIN {X 0,Y 566.222,Z 647.771,A -85,B 0,C 180,E1 -2401.859,E2 -2401.859} C_VEL
LIN {X 0,Y 566.208,Z 647.768,A -85,B 0,C 180,E1 -2404.251,E2 -2404.251} C_VEL
LIN {X 0,Y 566.186,Z 647.767,A -85,B 0,C 180,E1 -2406.714,E2 -2406.714} C_VEL
LIN {X 0,Y 566.209,Z 647.765,A -85,B 0,C 180,E1 -2409.663,E2 -2409.663} C_VEL
LIN {X 0,Y 566.195,Z 647.768,A -85,B 0,C 180,E1 -2412.669,E2 -2412.669} C_VEL
LIN {X 0,Y 566.229,Z 647.761,A -85,B 0,C 180,E1 -2415.627,E2 -2415.627} C_VEL
LIN {X 0,Y 566.23,Z 647.769,A -85,B 0,C 180,E1 -2418.675,E2 -2418.675} C_VEL
LIN {X 0,Y 566.229,Z 647.76,A -85,B 0,C 180,E1 -2421.435,E2 -2421.435} C_VEL
LIN {X 0,Y 566.257,Z 647.76,A -85,B 0,C 180,E1 -2424.302,E2 -2424.302} C_VEL
LIN {X 0,Y 566.279,Z 647.754,A -85,B 0,C 180,E1 -2427.866,E2 -2427.866} C_VEL
LIN {X 0,Y 566.297,Z 647.757,A -85,B 0,C 180,E1 -2430.711,E2 -2430.711} C_VEL
LIN {X 0,Y 566.268,Z 647.761,A -85,B 0,C 180,E1 -2432.846,E2 -2432.846} C_VEL
LIN {X 0,Y 566.257,Z 647.76,A -85,B 0,C 180,E1 -2435.698,E2 -2435.698} C_VEL
LIN {X 0,Y 566.229,Z 647.76,A -85,B 0,C 180,E1 -2438.565,E2 -2438.565} C_VEL
LIN {X 0,Y 566.238,Z 647.768,A -85,B 0,C 180,E1 -2441.454,E2 -2441.454} C_VEL
LIN {X 0,Y 566.23,Z 647.76,A -85,B 0,C 180,E1 -2444.506,E2 -2444.506} C_VEL
LIN {X 0,Y 566.195,Z 647.768,A -85,B 0,C 180,E1 -2447.331,E2 -2447.331} C_VEL
LIN {X 0,Y 566.209,Z 647.765,A -85,B 0,C 180,E1 -2450.337,E2 -2450.337} C_VEL
LIN {X 0,Y 566.184,Z 647.768,A -85,B 0,C 180,E1 -2453.403,E2 -2453.403} C_VEL
LIN {X 0,Y 566.208,Z 647.768,A -85,B 0,C 180,E1 -2455.749,E2 -2455.749} C_VEL
LIN {X 0,Y 566.2,Z 647.773,A -85,B 0,C 180,E1 -2458.202,E2 -2458.202} C_VEL
LIN {X 0,Y 566.188,Z 647.77,A -85,B 0,C 180,E1 -2460.591,E2 -2460.591} C_VEL
LIN {X 0,Y 566.222,Z 647.761,A -85,B 0,C 180,E1 -2463.101,E2 -2463.101} C_VEL
LIN {X 0,Y 566.204,Z 647.763,A -85,B 0,C 180,E1 -2465.688,E2 -2465.688} C_VEL
LIN {X 0,Y 566.207,Z 647.772,A -85,B 0,C 180,E1 -2468.558,E2 -2468.558} C_VEL
LIN {X 0,Y 566.203,Z 647.766,A -85,B 0,C 180,E1 -2471.136,E2 -2471.136} C_VEL
LIN {X 0,Y 566.191,Z 647.765,A -85,B 0,C 180,E1 -2474.035,E2 -2474.035} C_VEL
LIN {X 0,Y 566.205,Z 647.771,A -85,B 0,C 180,E1 -2477.081,E2 -2477.081} C_VEL
LIN {X 0,Y 566.218,Z 647.761,A -85,B 0,C 180,E1 -2479.802,E2 -2479.802} C_VEL
LIN {X 0,Y 566.189,Z 647.765,A -85,B 0,C 180,E1 -2482.598,E2 -2482.598} C_VEL
LIN {X 0,Y 566.213,Z 647.765,A -85,B 0,C 180,E1 -2485.183,E2 -2485.183} C_VEL
LIN {X 0,Y 566.225,Z 647.763,A -85,B 0,C 180,E1 -2487.744,E2 -2487.744} C_VEL
LIN {X 0,Y 566.218,Z 647.754,A -85,B 0,C 180,E1 -2490.323,E2 -2490.323} C_VEL
LIN {X 0,Y 566.224,Z 647.762,A -85,B 0,C 180,E1 -2493.335,E2 -2493.335} C_VEL
LIN {X 0,Y 566.194,Z 647.771,A -85,B 0,C 180,E1 -2495.819,E2 -2495.819} C_VEL
LIN {X 0,Y 566.206,Z 647.761,A -85,B 0,C 180,E1 -2498.903,E2 -2498.903} C_VEL
LIN {X 0,Y 566.203,Z 647.763,A -85,B 0,C 180,E1 -2501.173,E2 -2501.173} C_VEL
LIN {X 0,Y 566.211,Z 647.762,A -85,B 0,C 180,E1 -2503.413,E2 -2503.413} C_VEL
LIN {X 0,Y 566.19,Z 647.767,A -85,B 0,C 180,E1 -2506.359,E2 -2506.359} C_VEL
LIN {X 0,Y 566.263,Z 647.757,A -85,B 0,C 180,E1 -2508.654,E2 -2508.654} C_VEL
LIN {X 0,Y 566.238,Z 647.756,A -85,B 0,C 180,E1 -2511.435,E2 -2511.435} C_VEL
LIN {X 0,Y 566.26,Z 647.763,A -85,B 0,C 180,E1 -2514.302,E2 -2514.302} C_VEL
LIN {X 0,Y 566.271,Z 647.752,A -85,B 0,C 180,E1 -2517.866,E2 -2517.866} C_VEL
LIN {X 0,Y 566.3,Z 647.76,A -85,B 0,C 180,E1 -2520.711,E2 -2520.711} C_VEL
LIN {X 0,Y 566.271,Z 647.761,A -85,B 0,C 180,E1 -2522.846,E2 -2522.846} C_VEL
LIN {X 0,Y 566.26,Z 647.755,A -85,B 0,C 180,E1 -2525.698,E2 -2525.698} C_VEL
LIN {X 0,Y 566.239,Z 647.758,A -85,B 0,C 180,E1 -2528.566,E2 -2528.566} C_VEL
LIN {X 0,Y 566.24,Z 647.761,A -85,B 0,C 180,E1 -2531.454,E2 -2531.454} C_VEL
LIN {X 0,Y 566.223,Z 647.759,A -85,B 0,C 180,E1 -2534.508,E2 -2534.508} C_VEL
LIN {X 0,Y 566.194,Z 647.771,A -85,B 0,C 180,E1 -2537.332,E2 -2537.332} C_VEL
LIN {X 0,Y 566.21,Z 647.762,A -85,B 0,C 180,E1 -2540.337,E2 -2540.337} C_VEL
LIN {X 0,Y 566.181,Z 647.77,A -85,B 0,C 180,E1 -2543.404,E2 -2543.404} C_VEL
LIN {X 0,Y 566.218,Z 647.768,A -85,B 0,C 180,E1 -2545.749,E2 -2545.749} C_VEL
LIN {X 0,Y 566.198,Z 647.757,A -85,B 0,C 180,E1 -2548.204,E2 -2548.204} C_VEL
LIN {X 0,Y 566.185,Z 647.764,A -85,B 0,C 180,E1 -2550.593,E2 -2550.593} C_VEL
LIN {X 0,Y 566.22,Z 647.76,A -85,B 0,C 180,E1 -2553.102,E2 -2553.102} C_VEL
LIN {X 0,Y 566.205,Z 647.762,A -85,B 0,C 180,E1 -2555.689,E2 -2555.689} C_VEL
LIN {X 0,Y 566.211,Z 647.766,A -85,B 0,C 180,E1 -2558.56,E2 -2558.56} C_VEL
LIN {X 0,Y 566.214,Z 647.757,A -85,B 0,C 180,E1 -2561.136,E2 -2561.136} C_VEL
LIN {X 0,Y 566.194,Z 647.768,A -85,B 0,C 180,E1 -2564.036,E2 -2564.036} C_VEL
LIN {X 0,Y 566.198,Z 647.766,A -85,B 0,C 180,E1 -2567.083,E2 -2567.083} C_VEL
LIN {X 0,Y 566.221,Z 647.76,A -85,B 0,C 180,E1 -2569.803,E2 -2569.803} C_VEL
LIN {X 0,Y 566.194,Z 647.764,A -85,B 0,C 180,E1 -2572.6,E2 -2572.6} C_VEL
LIN {X 0,Y 566.216,Z 647.769,A -85,B 0,C 180,E1 -2575.184,E2 -2575.184} C_VEL
LIN {X 0,Y 566.232,Z 647.749,A -85,B 0,C 180,E1 -2577.744,E2 -2577.744} C_VEL
LIN {X 0,Y 566.274,Z 647.961,A -85,B 0,C 180,E1 -2579.373,E2 -2579.373} C_VEL
LIN {X 0,Y 568.231,Z 656.786,A -85,B 0,C 180,E1 -2580.756,E2 -2580.756} C_VEL
LIN {X 0,Y 567.842,Z 677.192,A -85,B 0,C 180,E1 -2583.542,E2 -2583.542} C_VEL
LIN {X 0,Y 567.567,Z 695.928,A -85,B 0,C 180,E1 -2586.024,E2 -2586.024} C_VEL
LIN {X 0,Y 569.646,Z 704.675,A -85,B 0,C 180,E1 -2586.256,E2 -2586.256} C_VEL
LIN {X 0,Y 568.925,Z 895.959,A -85,B 0,C 180,E1 -2588.795,E2 -2588.795} C_VEL
LIN {X 0,Y 568.752,Z 911.404,A -85,B 0,C 180,E1 -2589.096,E2 -2589.096} C_VEL
LIN {X 0,Y 568.578,Z 925.654,A -85,B 0,C 180,E1 -2589.492,E2 -2589.492} C_VEL
LIN {X 0,Y 568.316,Z 940.555,A -85,B 0,C 180,E1 -2590.025,E2 -2590.025} C_VEL
LIN {X 0,Y 567.998,Z 956.806,A -85,B 0,C 180,E1 -2590.766,E2 -2590.766} C_VEL
LIN {X 0,Y 567.674,Z 971.531,A -85,B 0,C 180,E1 -2591.598,E2 -2591.598} C_VEL
LIN {X 0,Y 567.37,Z 985.096,A -85,B 0,C 180,E1 -2592.515,E2 -2592.515} C_VEL
LIN {X 0,Y 567.064,Z 997.905,A -85,B 0,C 180,E1 -2593.531,E2 -2593.531} C_VEL
LIN {X 0,Y 566.829,Z 1008.888,A -85,B 0,C 180,E1 -2594.54,E2 -2594.54} C_VEL
LIN {X 0,Y 566.599,Z 1020.891,A -85,B 0,C 180,E1 -2595.82,E2 -2595.82} C_VEL
LIN {X 0,Y 566.34,Z 1032.423,A -85,B 0,C 180,E1 -2597.276,E2 -2597.276} C_VEL
LIN {X 0,Y 566.204,Z 1041.825,A -85,B 0,C 180,E1 -2598.691,E2 -2598.691} C_VEL
LIN {X 0,Y 566.085,Z 1049.21,A -85,B 0,C 180,E1 -2599.991,E2 -2599.991} C_VEL
LIN {X 0,Y 566.023,Z 1056.083,A -85,B 0,C 180,E1 -2601.431,E2 -2601.431} C_VEL
LIN {X 0,Y 565.966,Z 1061.734,A -85,B 0,C 180,E1 -2602.867,E2 -2602.867} C_VEL
LIN {X 0,Y 565.961,Z 1066.234,A -85,B 0,C 180,E1 -2604.299,E2 -2604.299} C_VEL
LIN {X 0,Y 565.91,Z 1069.65,A -85,B 0,C 180,E1 -2605.727,E2 -2605.727} C_VEL
LIN {X 0,Y 565.866,Z 1072.084,A -85,B 0,C 180,E1 -2607.152,E2 -2607.152} C_VEL
LIN {X 0,Y 565.841,Z 1073.494,A -85,B 0,C 180,E1 -2608.577,E2 -2608.577} C_VEL
LIN {X 0,Y 565.834,Z 1074,A -85,B 0,C 180,E1 -2610,E2 -2610} C_VEL
LIN {X 0,Y 565.841,Z 1073.494,A -85,B 0,C 180,E1 -2611.423,E2 -2611.423} C_VEL
LIN {X 0,Y 565.866,Z 1072.084,A -85,B 0,C 180,E1 -2612.848,E2 -2612.848} C_VEL
LIN {X 0,Y 565.911,Z 1069.65,A -85,B 0,C 180,E1 -2614.273,E2 -2614.273} C_VEL
LIN {X 0,Y 565.913,Z 1065.173,A -85,B 0,C 180,E1 -2616.059,E2 -2616.059} C_VEL
LIN {X 0,Y 565.97,Z 1060.431,A -85,B 0,C 180,E1 -2617.492,E2 -2617.492} C_VEL
LIN {X 0,Y 566.012,Z 1054.474,A -85,B 0,C 180,E1 -2618.929,E2 -2618.929} C_VEL
LIN {X 0,Y 566.125,Z 1046.293,A -85,B 0,C 180,E1 -2620.551,E2 -2620.551} C_VEL
LIN {X 0,Y 566.245,Z 1037.449,A -85,B 0,C 180,E1 -2621.999,E2 -2621.999} C_VEL
LIN {X 0,Y 566.409,Z 1028.331,A -85,B 0,C 180,E1 -2623.27,E2 -2623.27} C_VEL
LIN {X 0,Y 566.61,Z 1017.895,A -85,B 0,C 180,E1 -2624.517,E2 -2624.517} C_VEL
LIN {X 0,Y 566.853,Z 1006.992,A -85,B 0,C 180,E1 -2625.644,E2 -2625.644} C_VEL
LIN {X 0,Y 567.143,Z 994.657,A -85,B 0,C 180,E1 -2626.745,E2 -2626.745} C_VEL
LIN {X 0,Y 567.498,Z 979.94,A -85,B 0,C 180,E1 -2627.856,E2 -2627.856} C_VEL
LIN {X 0,Y 567.826,Z 965.314,A -85,B 0,C 180,E1 -2628.771,E2 -2628.771} C_VEL
LIN {X 0,Y 568.104,Z 951.026,A -85,B 0,C 180,E1 -2629.512,E2 -2629.512} C_VEL
LIN {X 0,Y 568.397,Z 937.795,A -85,B 0,C 180,E1 -2630.081,E2 -2630.081} C_VEL
LIN {X 0,Y 568.6,Z 923.419,A -85,B 0,C 180,E1 -2630.578,E2 -2630.578} C_VEL
LIN {X 0,Y 568.794,Z 907.481,A -85,B 0,C 180,E1 -2630.997,E2 -2630.997} C_VEL
LIN {X 0,Y 568.985,Z 887.835,A -85,B 0,C 180,E1 -2631.321,E2 -2631.321} C_VEL
LIN {X 0,Y 569.676,Z 705.297,A -85,B 0,C 180,E1 -2633.734,E2 -2633.734} C_VEL
